// TwinCAT 3 PLC project Plc_Program
// ProgramVersion: 3.1.4026.15
// libraries:
//   CPNTeck - OSCAT BASIC, * (CPNTeck - Automação Industrial)
//   Tc2_MC2, * (Beckhoff Automation GmbH)
//   Tc2_ModbusSrv, * (Beckhoff Automation GmbH)
//   Tc2_Standard, * (Beckhoff Automation GmbH)
//   Tc2_SUPS, * (Beckhoff Automation GmbH)
//   Tc2_System, * (Beckhoff Automation GmbH)
//   Tc2_Utilities, * (Beckhoff Automation GmbH)
// project tree:
//   GVLs/ GVL_Hmi.TcGVL, GVL_Hw.TcGVL, GVL_InterConnection.TcGVL
//   Library/AxisControl/DataTypes/ LAxisCtrl_typeAxisConfig.TcDUT, LAxisCtrl_typeCamIn.TcDUT, LAxisCtrl_typeDiagnostics.TcDUT, LAxisCtrl_typeFastStop.TcDUT, LAxisCtrl_typeGearInAbsolute.TcDUT, LAxisCtrl_typeGearInRelative.TcDUT, LAxisCtrl_typeGeneralSettings.TcDUT, LAxisCtrl_typeHoming.TcDUT, LAxisCtrl_typeJog.TcDUT, LAxisCtrl_typeMoveVelocity.TcDUT, LAxisCtrl_typePhasing.TcDUT, LAxisCtrl_typePosAbsolute.TcDUT, LAxisCtrl_typePosRelative.TcDUT, LAxisCtrl_typePosSuperimposed.TcDUT, LAxisCtrl_typePower.TcDUT, LAxisCtrl_typeStop.TcDUT, LAxisCtrl_typeTorqueLimiting.TcDUT, LRK_typeCamCommand.TcDUT, LRK_typeCamStatus.TcDUT, LRK_typeRotaryKnifeAxisCommand.TcDUT, LRK_typeUsersInterface.TcDUT, MC_SYNCHRONIZEDMOTIONSIMULATION.TcPOU, TO_Cam_Struct_PointData.TcDUT, TO_Cam_Struct_SegmentData.TcDUT
//   Library/AxisControl/ FB_ComplexAxisControl.TcPOU (excluded from build), FB_SimpleAxisControl.TcPOU, MC_TORQUELIMITING.TcPOU
//   Library/Beckhoff/CX9020/ FB_SavePersistentData.TcPOU
//   Library/Beckhoff/EL1008/DataTypes/ EL1008_DEV_CONFIG.TcDUT, EL1008_HWTOPLC_PDOS.TcDUT, EL1008_PDOS.TcDUT
//   Library/Beckhoff/EL1008/ FB_EL1008.TcPOU
//   Library/Beckhoff/EL1809/DataTypes/ EL1809_DEV_CONFIG.TcDUT, EL1809_HWTOPLC_PDOS.TcDUT, EL1809_PDOS.TcDUT
//   Library/Beckhoff/EL1809/ FB_EL1809.TcPOU
//   Library/Beckhoff/EL2809/DataTypes/ EL2809_DEV_CONFIG.TcDUT, EL2809_PDOS.TcDUT, EL2809_PLCTOHW_PDOS.TcDUT
//   Library/Beckhoff/EL2809/ FB_EL2809.TcPOU
//   Library/Beckhoff/EL3002 - Ai 2 x 10V - 12bit/DataTypes/ EL3002_CHANNEL.TcDUT, EL3002_DEV_CONFIG.TcDUT, EL3002_DEV_STATUS.TcDUT, EL3002_HWTOPLC_PDOS.TcDUT, EL3002_PDOS.TcDUT
//   Library/Beckhoff/EL3002 - Ai 2 x 10V - 12bit/ FB_EL3002.TcPOU
//   Library/Beckhoff/EL4004 - AQ 4 x 0-10V/DataTypes/ EL4004_DEV_CONFIG.TcDUT, EL4004_HWTOPLC_PDOS.TcDUT, EL4004_PDOS.TcDUT
//   Library/Beckhoff/EL4004 - AQ 4 x 0-10V/ FB_EL4004.TcPOU
//   Library/Beckhoff/EL5152 -2 x  Encoder Input/DataTypes/ EL5152_CONTROL.TcDUT, EL5152_DEV_CONFIG.TcDUT, EL5152_HWTOPLC.TcDUT, EL5152_HWTOPLC_PDOS.TcDUT, EL5152_PLCTOHW.TcDUT, EL5152_PLCTOHW_PDOS.TcDUT, EL5152_STATUS.TcDUT
//   Library/Beckhoff/EL5152 -2 x  Encoder Input/ FB_EL5152.TcPOU
//   Library/EL6910 - TwinSAFE PLC/ EL6910_ESTOP.TcDUT, EL6910_ESTOP_DIGNOSTICS.TcDUT, EL6910_ESTOP_STATUS.TcDUT, EL6910_HWTOPLC_PDOS.TcDUT, EL6910_PDOS.TcDUT, EL6910_PLCTOHW_PDOS.TcDUT, FB_EL6910.TcPOU
//   Library/FAS/IO-Link/006B51 - IO-Link Master/DataTypes/ _006B51_Channel_State.TcDUT, _006B51_HWTOPLC_PDOS.TcDUT
//   Library/FAS/IO-Link/006B51 - IO-Link Master/ _FB_006B51.TcPOU
//   Library/FAS/IO-Link/00BE31 - IP67 16Di or 16Do/DataTypes/ _00BE31_HWTOPLC_PDOS.TcDUT, _00BE31_PLCTOHW_PDOS.TcDUT
//   Library/FAS/IO-Link/00BE31 - IP67 16Di or 16Do/ _FB_00BE31.TcPOU
//   Library/FAS/IO-Link/00BH11 - 16Di or 16Do/DataTypes/ _00BH11_HWTOPLC_PDOS.TcDUT, _00BH11_PLCTOHW_PDOS.TcDUT
//   Library/FAS/IO-Link/00BH11 - 16Di or 16Do/ _FB_00BH11.TcPOU
//   Library/FAS/IO-Link/00BW12 - 16 Solenoid Island/DataTypes/ _00BW12_PLCTOHW_PDOS.TcDUT
//   Library/FAS/IO-Link/00BW12 - 16 Solenoid Island/ _FB_00BW1.TcPOU
//   Library/FAS/IO-Link/0AC001 - Analog Input/DataTypes/ _0AC001_DEV_CONFIG.TcDUT, _0AC001_HWTOPLC_PDOS.TcDUT
//   Library/FAS/IO-Link/0AC001 - Analog Input/ _FB_0AC001.TcPOU
//   Library/Machine/DryEnd/Alarm Control/ FB_AlarmControl.TcPOU
//   Library/Machine/DryEnd/AutomaticOrderChange/ aocConfig_TypeStruct.TcDUT, aocHmiCommands_TypeStruct.TcDUT, aocHmiStatus_TypeStruct.TcDUT, FB_AutomaticOrderChange.TcPOU, FB_AutomaticOrderChange_V1.TcPOU, FB_AutomaticOrderChange_V1_BAK.TcPOU, lineControlHmiCommands_TypeStruct.TcDUT
//   Library/Machine/DryEnd/Hmi/ hmiAlarms_TypeStruct.TcDUT, hmiCommands_TypeStruct.TcDUT, hmiStatus_TypeStruct.TcDUT, machineConfig_TypeStruct.TcDUT
//   Library/Machine/DryEnd/Order control/DataTypes/ generatedOrderStatusWord_TypeStruct.TcDUT, generatedOrder_TypeStruct.TcDUT, orderConfig_TypeStruct.TcDUT, orderHmiCommands_TypeStruct.TcDUT, orderHmiStatus_TypeStruct.TcDUT, orderVariables_TypeStruct.TcDUT, order_TypeStruct.TcDUT, sheetTypeEnum.TcDUT
//   Library/Machine/DryEnd/Order control/ FB_MetricsAndCalculation.TcPOU
//   Library/Machine/Rotary knife/Config/ rotaryKnifeConfig_TypeStruct.TcDUT, rotaryKnifeHmiStatus_TypeStruct.TcDUT, rotaryKnifeSpeedCurve_TypeConfig.TcDUT, rotaryKnifeStatusWord1_TypeStruct.TcDUT, rotaryKnifeStatusWord2_TypeStruct.TcDUT
//   Library/Machine/Rotary knife/Function Block/ FB_RotaryKnife.TcPOU, FB_RotaryKnife_1.TcPOU, FB_SpeedLimit.TcPOU
//   Library/Machine/Rotary knife/Hmi/ hmiAlarmsRotaryKnife_TypeStruct.TcDUT, rotaryKnifeCommands_TypeStruct.TcDUT, rotaryKnifeStatus_TypeStruct.TcDUT
//   Library/Machine/Slitter/DataTypes/Hmi/ E_LevelSelector.TcDUT, hmiAlarmsSlitter_TypeStruct.TcDUT, hmiCommandsFlaps_TypeStruct.TcDUT, hmiCommandsJog_TypeStruct.TcDUT, hmiCommandsSmallPosCorrection_TypeStruct.TcDUT, hmiSlitterAlarms_TypeStruct.TcDUT, slitterCommands_TypeStruct.TcDUT, slitterConfig_TypeStruct.TcDUT, slitterStatus_TypeStruct.TcDUT
//   Library/Machine/Slitter/FunctionBlocks/ FB_KnifeLubrification.TcPOU, FB_KnifeSharpening.TcPOU, FB_KnifeSharpening_old.TcPOU, FB_PaperDirectionControl.TcPOU, FB_PaperDirectionControl_.TcPOU, FB_PositionsGeneration.TcPOU, FB_ScorerHeight.TcPOU, FB_SlitterControl.TcPOU, FB_SpeedMeter.TcPOU
//   Library/Machine/Stacker/Cpx/ FB_ComplexSheetStackerControl_1.TcPOU, FB_ComplexSheetStackerControl.TcPOU
//   Library/Machine/Stacker/Simple/DataTypes/ hmiAlarmsSimpleStacker_TypeStruct.TcDUT, hmiCommandsSimpleStacker_TypeStruct.TcDUT, hmiStatusSimpleStacker_TypeStruct.TcDUT, SimpleStackerConfig_TypeStruct.TcDUT, SimpleStackerConfig_TypeStruct_1.TcDUT
//   Library/Machine/Stacker/Cpx/DataTypes/ ComplexStackerConfig_TypeStruct.TcDUT, hmiAlarmsComplexStacker_TypeStruct.TcDUT, hmiCommandsComplexStacker_TypeStruct.TcDUT, hmiStatusComplexStacker_TypeStruct.TcDUT
//   Library/Machine/Stacker/Simple/ E_BackstopState.TcDUT, E_ConveyorLevelerState.TcDUT, E_PackageSeparationState.TcDUT, E_SheetStackDischargeState.TcDUT, E_SyncConveyorsState.TcDUT, FB_SimpleSheetStackerControl.TcPOU, FB_SimpleSheetStackerControl_1.TcPOU, FB_SimpleSheetStackerControl_2.TcPOU (not stored), FB_SimpleSheetStackerControl_3.TcPOU
//   Library/Ramp/ FB_Gen_SRamp.TcPOU
//   Library/Sick/DT35-B15251 - Laser Sensor/DataTypes/ _DT35B15251_DEV_CONFIG.TcDUT, _DT35B15251_HWTOPLC_PDOS.TcDUT
//   Library/Sick/DT35-B15251 - Laser Sensor/ _FB_DT35_B15251.TcPOU
//   Library/Inovance/IS620P-CO/DataTypes/ E_IS620P_CO_STATE.TcDUT, IS620P_CO_DEV_CONFIG.TcDUT, IS620P_CO_HWTOPLC_PDOS.TcDUT, IS620P_CO_PLCTOHW_PDOS.TcDUT, IS620P_CO_STATUS.TcDUT
//   Library/Inovance/IS620P-CO/FB/ FB_IS620P_CO.TcPOU
//   / PlcFastTask.TcTTO, PlcTask.TcTTO, RecipeManager.TcRMO (not stored)
//   POUs/ FAST.TcPOU, MAIN.TcPOU
// real-time tasks:
//   TASK PlcTask: cycle T#20ms, priority 20, ADS port 350
//   TASK PlcFastTask: cycle T#5ms, priority 1, ADS port 351
// motion (NC):
//   TASK NC-Task 1 SAF: cycle T#4ms, priority 4, ADS port 501
//   TASK NC-Task 1 SVB: cycle T#10ms, priority 8, ADS port 511
//   AXIS knife1_Axis (id 1)
//     Velo: RefSearch=20, RefSync=2
//     PositionAreaControl: Enable=false
//     OtherSettings: AllowMotionCmdToSlave=true
//     encoder EncType=19
//       EncPara: ScaleFactorNumerator=5.96046448e-07, ModuloFactor=5, Inverse=true, MaxCount=#xffffffff
//         SoftEndMinControl: Enable=true
//         SoftEndMaxControl: Enable=true, Range=950
//         Inc: RefSearchInverse=true, RefSyncInverse=false
//     drive DrvType=16
//       DrvPara: Inverse=true, MaxCount=#xffffffff, DriveControlDWord=#x00020000
//         Analog: TorqueSetpointScale=10, ScaleFactorActTorque=0.1
//         TimeComp: TaskDelayCycles=1
//     controller CtrType=1
//       CtrPara: PriorControlFactor=1
//         PosDiffControl: Enable=false
//         Observer: BandWidth=20
//   AXIS knife2_Axis (id 2)
//     Velo: RefSearch=20, RefSync=2
//     PositionAreaControl: Enable=false
//     OtherSettings: AllowMotionCmdToSlave=true
//     encoder EncType=19
//       EncPara: ScaleFactorNumerator=5.96046448e-07, ModuloFactor=5, Inverse=true, MaxCount=#xffffffff
//         SoftEndMinControl: Enable=true
//         SoftEndMaxControl: Enable=true, Range=1080
//         Inc: RefSearchInverse=true, RefSyncInverse=false
//     drive DrvType=16
//       DrvPara: Inverse=true, MaxCount=#xffffffff, DriveControlDWord=#x00020000
//         Analog: TorqueSetpointScale=10, ScaleFactorActTorque=0.1
//         TimeComp: TaskDelayCycles=1
//     controller CtrType=1
//       CtrPara: PriorControlFactor=1
//         PosDiffControl: Enable=false
//         Observer: BandWidth=20
//   AXIS knife3_Axis (id 3)
//     Velo: RefSearch=20, RefSync=2
//     PositionAreaControl: Enable=false
//     OtherSettings: AllowMotionCmdToSlave=true
//     encoder EncType=19
//       EncPara: ScaleFactorNumerator=5.96046448e-07, ModuloFactor=5, Inverse=true, MaxCount=#xffffffff
//         SoftEndMinControl: Enable=true
//         SoftEndMaxControl: Enable=true, Range=1220
//         Inc: RefSearchInverse=true, RefSyncInverse=false
//     drive DrvType=16
//       DrvPara: Inverse=true, MaxCount=#xffffffff, DriveControlDWord=#x00020000
//         Analog: TorqueSetpointScale=10, ScaleFactorActTorque=0.1
//         TimeComp: TaskDelayCycles=1
//     controller CtrType=1
//       CtrPara: PriorControlFactor=1
//         PosDiffControl: Enable=false
//         Observer: BandWidth=20
//   AXIS knife4_Axis (id 4)
//     Velo: RefSearch=20, RefSync=2
//     PositionAreaControl: Enable=false
//     OtherSettings: AllowMotionCmdToSlave=true
//     encoder EncType=19
//       EncPara: ScaleFactorNumerator=5.96046448e-07, ModuloFactor=5, MaxCount=#xffffffff
//         SoftEndMinControl: Enable=true, Range=1176
//         SoftEndMaxControl: Enable=true, Range=3000
//     drive DrvType=16
//       DrvPara: MaxCount=#xffffffff, DriveControlDWord=#x00020000
//         Analog: TorqueSetpointScale=10, ScaleFactorActTorque=0.1
//         TimeComp: TaskDelayCycles=1
//     controller CtrType=1
//       CtrPara: PriorControlFactor=1
//         PosDiffControl: Enable=false
//         Observer: BandWidth=20
//   AXIS knife5_Axis (id 5)
//     Velo: RefSearch=20, RefSync=2
//     PositionAreaControl: Enable=false
//     OtherSettings: AllowMotionCmdToSlave=true
//     encoder EncType=19
//       EncPara: ScaleFactorNumerator=5.96046448e-07, ModuloFactor=5, MaxCount=#xffffffff
//         SoftEndMinControl: Enable=true, Range=1300
//         SoftEndMaxControl: Enable=true, Range=3000
//     drive DrvType=16
//       DrvPara: MaxCount=#xffffffff, DriveControlDWord=#x00020000
//         Analog: TorqueSetpointScale=10, ScaleFactorActTorque=0.1
//         TimeComp: TaskDelayCycles=1
//     controller CtrType=1
//       CtrPara: PriorControlFactor=1
//         PosDiffControl: Enable=false
//         Observer: BandWidth=20
//   AXIS Scorer1_Axis (id 6)
//     Velo: RefSearch=20, RefSync=2
//     PositionAreaControl: Enable=false
//     OtherSettings: AllowMotionCmdToSlave=true
//     encoder EncType=19
//       EncPara: ScaleFactorNumerator=5.96046448e-07, ModuloFactor=5, Inverse=true, MaxCount=#xffffffff
//         SoftEndMaxControl: Range=968
//         Inc: RefSearchInverse=true, RefSyncInverse=false
//     drive DrvType=16
//       DrvPara: Inverse=true, MaxCount=#xffffffff, DriveControlDWord=#x00020000
//         Analog: TorqueSetpointScale=10, ScaleFactorActTorque=0.1
//         TimeComp: TaskDelayCycles=1
//     controller CtrType=1
//       CtrPara: PriorControlFactor=1
//         PosDiffControl: Enable=false
//         Observer: BandWidth=20
//   AXIS Scorer2_Axis (id 7)
//     Velo: RefSearch=20, RefSync=2
//     PositionAreaControl: Enable=false
//     OtherSettings: AllowMotionCmdToSlave=true
//     encoder EncType=19
//       EncPara: ScaleFactorNumerator=5.96046448e-07, ModuloFactor=5, Inverse=true, MaxCount=#xffffffff
//         SoftEndMaxControl: Range=968
//         Inc: RefSearchInverse=true, RefSyncInverse=false
//     drive DrvType=16
//       DrvPara: Inverse=true, MaxCount=#xffffffff, DriveControlDWord=#x00020000
//         Analog: TorqueSetpointScale=10, ScaleFactorActTorque=0.1
//         TimeComp: TaskDelayCycles=1
//     controller CtrType=1
//       CtrPara: PriorControlFactor=1
//         PosDiffControl: Enable=false
//         Observer: BandWidth=20
//   AXIS Scorer3_Axis (id 8)
//     Velo: RefSearch=20, RefSync=2
//     PositionAreaControl: Enable=false
//     OtherSettings: AllowMotionCmdToSlave=true
//     encoder EncType=19
//       EncPara: ScaleFactorNumerator=5.96046448e-07, ModuloFactor=5, Inverse=true, MaxCount=#xffffffff
//         SoftEndMinControl: Range=364
//         SoftEndMaxControl: Range=1120
//         Inc: RefSearchInverse=true, RefSyncInverse=false
//     drive DrvType=16
//       DrvPara: Inverse=true, MaxCount=#xffffffff, DriveControlDWord=#x00020000
//         Analog: TorqueSetpointScale=10, ScaleFactorActTorque=0.1
//         TimeComp: TaskDelayCycles=1
//     controller CtrType=1
//       CtrPara: PriorControlFactor=1
//         PosDiffControl: Enable=false
//         Observer: BandWidth=20
//   AXIS Scorer4_Axis (id 9)
//     Velo: RefSearch=20, RefSync=2
//     PositionAreaControl: Enable=false
//     OtherSettings: AllowMotionCmdToSlave=true
//     encoder EncType=19
//       EncPara: ScaleFactorNumerator=5.96046448e-07, ModuloFactor=5, Inverse=true, MaxCount=#xffffffff
//         SoftEndMinControl: Range=340
//         SoftEndMaxControl: Range=1120
//         Inc: RefSearchInverse=true, RefSyncInverse=false
//     drive DrvType=16
//       DrvPara: Inverse=true, MaxCount=#xffffffff, DriveControlDWord=#x00020000
//         Analog: TorqueSetpointScale=10, ScaleFactorActTorque=0.1
//         TimeComp: TaskDelayCycles=1
//     controller CtrType=1
//       CtrPara: PriorControlFactor=1
//         PosDiffControl: Enable=false
//         Observer: BandWidth=20
//   AXIS Scorer5_Axis (id 10)
//     Velo: RefSearch=20, RefSync=2
//     PositionAreaControl: Enable=false
//     OtherSettings: AllowMotionCmdToSlave=true
//     encoder EncType=19
//       EncPara: ScaleFactorNumerator=5.96046448e-07, ModuloFactor=5, MaxCount=#xffffffff
//         SoftEndMinControl: Range=1050
//         SoftEndMaxControl: Range=1846
//     drive DrvType=16
//       DrvPara: MaxCount=#xffffffff, DriveControlDWord=#x00020000
//         Analog: TorqueSetpointScale=10, ScaleFactorActTorque=0.1
//         TimeComp: TaskDelayCycles=1
//     controller CtrType=1
//       CtrPara: PriorControlFactor=1
//         PosDiffControl: Enable=false
//         Observer: BandWidth=20
//   AXIS Scorer6_Axis (id 11)
//     Velo: RefSearch=20, RefSync=2
//     PositionAreaControl: Enable=false
//     OtherSettings: AllowMotionCmdToSlave=true
//     encoder EncType=19
//       EncPara: ScaleFactorNumerator=5.96046448e-07, ModuloFactor=5, MaxCount=#xffffffff
//         SoftEndMinControl: Range=1130
//         SoftEndMaxControl: Range=1890
//     drive DrvType=16
//       DrvPara: MaxCount=#xffffffff, DriveControlDWord=#x00020000
//         Analog: TorqueSetpointScale=10, ScaleFactorActTorque=0.1
//         TimeComp: TaskDelayCycles=1
//     controller CtrType=1
//       CtrPara: PriorControlFactor=1
//         PosDiffControl: Enable=false
//         Observer: BandWidth=20
//   AXIS Scorer7_Axis (id 12)
//     Velo: RefSearch=20, RefSync=2
//     PositionAreaControl: Enable=false
//     OtherSettings: AllowMotionCmdToSlave=true
//     encoder EncType=19
//       EncPara: ScaleFactorNumerator=5.96046448e-07, ModuloFactor=5, MaxCount=#xffffffff
//         SoftEndMinControl: Range=1220
//         SoftEndMaxControl: Range=3000
//     drive DrvType=16
//       DrvPara: MaxCount=#xffffffff, DriveControlDWord=#x00020000
//         Analog: TorqueSetpointScale=10, ScaleFactorActTorque=0.1
//         TimeComp: TaskDelayCycles=1
//     controller CtrType=1
//       CtrPara: PriorControlFactor=1
//         PosDiffControl: Enable=false
//         Observer: BandWidth=20
//   AXIS Scorer8_Axis (id 13)
//     Velo: RefSearch=20, RefSync=2
//     PositionAreaControl: Enable=false
//     OtherSettings: AllowMotionCmdToSlave=true
//     encoder EncType=19
//       EncPara: ScaleFactorNumerator=5.96046448e-07, ModuloFactor=5, MaxCount=#xffffffff
//         SoftEndMinControl: Range=1240
//         SoftEndMaxControl: Range=3000
//     drive DrvType=16
//       DrvPara: MaxCount=#xffffffff, DriveControlDWord=#x00020000
//         Analog: TorqueSetpointScale=10, ScaleFactorActTorque=0.1
//         TimeComp: TaskDelayCycles=1
//     controller CtrType=1
//       CtrPara: PriorControlFactor=1
//         PosDiffControl: Enable=false, Range=20
//         Observer: BandWidth=20
// I/O:
//   DEVICE ETC, AmsNetId 192.168.30.79.2.1
//     SLT1+P1=050-BC1 [EK1200-5000 EtherCAT Power supply (2A E-Bus)]
//       SLT1+P1=050-DI1 [EL1809 16Ch. Dig. Input 24V, 3ms]
//       SLT1+P1=050-DI2 [EL1809 16Ch. Dig. Input 24V, 3ms]
//       SLT1+P1=050-DI3 [EL1809 16Ch. Dig. Input 24V, 3ms]
//       SLT1+P1=050-DI4 [EL1809 16Ch. Dig. Input 24V, 3ms]
//       SLT1+P1=050-DI5 [EL1809 16Ch. Dig. Input 24V, 3ms]
//       SLT1+P1=050-DO1 [EL1809 16Ch. Dig. Input 24V, 3ms]
//       SLT1+P1=050-DO2 [EL2809 16Ch. Dig. Output 24V, 0.5A]
//       SLT1+P1=050-DO3 [EL2809 16Ch. Dig. Output 24V, 0.5A]
//       SLT1+P1=050-DO4 [EL2809 16Ch. Dig. Output 24V, 0.5A]
//       SLT1+P1=050-DO5 [EL2809 16Ch. Dig. Output 24V, 0.5A]
//       SLT1+P1=050-DO6 [EL2809 16Ch. Dig. Output 24V, 0.5A]
//       SLT1+P1=050-DO7 [EL2809 16Ch. Dig. Output 24V, 0.5A]
//       SLT1+P1=050-BC2 [EK1110 EtherCAT extension]
//     SLT1+P1=100-UG01 [SD700_ECAT_V1.2_G]
//     SLT1+P1=100-UG02 [SD700_ECAT_V1.2_G]
//     SLT1+P1=100-UG03 [SD700_ECAT_V1.2_G]
//     SLT1+P1=100-UG04 [SD700_ECAT_V1.2_G]
//     SLT1+P1=100-UG05 [SD700_ECAT_V1.2_G]
//     SLT1+P1=100-UG06 [SD700_ECAT_V1.2_G]
//     SLT1+P1=100-UG07 [SD700_ECAT_V1.2_G]
//     SLT1+P1=100-UG08 [SD700_ECAT_V1.2_G]
//     SLT1+P1=100-UG09 [SD700_ECAT_V1.2_G]
//     SLT1+P1=100-UG10 [SD700_ECAT_V1.2_G]
//     SLT1+P1=100-UG11 [SD700_ECAT_V1.2_G]
//     SLT1+P1=100-UG12 [SD700_ECAT_V1.2_G]
//     SLT1+P1=100-UG13 [SD700_ECAT_V1.2_G]
//     RK+P1=050-BC1 [EK1100 EtherCAT Coupler (2A E-Bus)]
//       RK+P1=050-DI1 [EL1809 16Ch. Dig. Input 24V, 3ms]
//       RK+P1=050-DI2 [EL1008 8Ch. Dig. Input 24V, 3ms]
//       RK+P1=050-DO1 [EL2809 16Ch. Dig. Output 24V, 0.5A]
//       RK+P1=050-DO2 [EL2809 16Ch. Dig. Output 24V, 0.5A]
//       RK+P1=050-AI1 [EL3002 2Ch. Ana. Input +/-10V]
//       RK+P1=050-AO1 [EL4004 4Ch. Ana. Output 0-10V, 12bit]
//       RK+P1=050-AO2 [EL4004 4Ch. Ana. Output 0-10V, 12bit] (disabled)
//       RK+P1=050-BE1 [EL9011 End Terminal]
//     STK+P2=050-BC1 [EK1100 EtherCAT Coupler (2A E-Bus)]
//       STK+P2=050-DI1 [EL1809 16Ch. Dig. Input 24V, 3ms]
//       STK+P2=050-DI2 [EL1809 16Ch. Dig. Input 24V, 3ms]
//       STK+P2=050-DO1 [EL2809 16Ch. Dig. Output 24V, 0.5A]
//       STK+P2=050-DO2 [EL2809 16Ch. Dig. Output 24V, 0.5A]
//       STK+P2=050-ENC1 [EL5152 2Ch. Inc. Encoder]
//       STK+P2=050-AO1 [EL4004 4Ch. Ana. Output 0-10V, 12bit]
//       STK+P2=050-AO2 [EL4004 4Ch. Ana. Output 0-10V, 12bit]
//       STK+P2=050-AO3 [EL4004 4Ch. Ana. Output 0-10V, 12bit]
//       STK+P2=050-AO4 [EL4004 4Ch. Ana. Output 0-10V, 12bit]
//       STK+P2=050-SP1 [EL6910, TwinSAFE PLC]
//       STK+P2=050-SI1 [EL1904, 4 Ch. Safety Input 24V, TwinSAFE]
//         modules: Module 1 (FSOES)
//       STK+P2=050-SI2 [EL1904, 4 Ch. Safety Input 24V, TwinSAFE]
//         modules: Module 1 (FSOES)
//       STK+P2=050-SO1 [EL2904, 4 Ch. Safety Output 24V, 0.5A, TwinSAFE]
//         modules: Module 1 (FSOES), Module 2 (DO)
//       STK+P2=050-BC2 [EL6751 CANopen Master]
//       STK+P2=050-BC3 [EK1110 EtherCAT extension]
//     STK+M=050-BC1 [FNI ECT-504-105-M]
//       modules: STKL+M=050-DIO1 - IO-Link slave IP67 [Machine drive side], STKL+M=050-DIO2  - IO-Link slave IP24 [Lower command box], STKL+M=050-BE1  - IO-Link Sick distance sensor [Backstop], STKU+M=050-DIO1  - IO-Link slave IP24 [Lower command box], STKU+M=050-DIO2  - IO-Link slave IP24 [Uppercommand box], STKU+M=050-DIO3  - IO-Link slave IP24 [Elevator drive side], Module 7 (Digital_IN), Module 8 (Digital_IN)
//   DEVICE Device 3 (NOV-DP-RAM)
//   DEVICE CANopen, AmsNetId 192.168.30.79.3.1
//     STK+P2=100-UG8 - Backstop Servo Drive
//     STK+P2=100-UG8 - Elevator Servo Drive
// variable links:
//   ETC <-> ETC/STK+P2=050-BC1/STK+P2=050-SI2
//     STK+P2=050-BC1/STK+P2=050-SP1/ConnectionOutputs/Message_4 RxPDO <-> Module 1 (FSOES)/TxPDO/FSOE
//   ETC <-> ETC/STK+P2=050-BC1/STK+P2=050-SO1
//     STK+P2=050-BC1/STK+P2=050-SP1/ConnectionOutputs/Message_5 RxPDO <-> Module 1 (FSOES)/TxPDO/FSOE
//   ETC <-> ETC/STK+P2=050-BC1/STK+P2=050-SP1
//     STK+P2=050-BC1/STK+P2=050-SI1/Module 1 (FSOES)/RxPDO/FSOE <-> ConnectionInputs/Message_3 TxPDO
//     STK+P2=050-BC1/STK+P2=050-SI2/Module 1 (FSOES)/RxPDO/FSOE <-> ConnectionInputs/Message_4 TxPDO
//     STK+P2=050-BC1/STK+P2=050-SI1/Module 1 (FSOES)/TxPDO/FSOE <-> ConnectionOutputs/Message_3 RxPDO
//     STK+P2=050-BC1/STK+P2=050-SO1/Module 1 (FSOES)/RxPDO/FSOE <-> ConnectionInputs/Message_5 TxPDO
//   NC-Task 1 SAF/Axes/Scorer1_Axis <-> ETC/SLT1+P1=100-UG06
//     Drive/Inputs/In/nDcOutputTime <-> InfoData/DcOutputShift
//     Drive/Inputs/In/nState1 <-> 2nd TxPDO Mapping/Status Word
//     Drive/Inputs/In/nState2 <-> 2nd TxPDO Mapping/Status Word @bit 8
//     Drive/Inputs/In/nState4 @bit 1 <-> WcState/InputToggle
//     Drive/Inputs/In/nState4 <-> WcState/WcState
//     Drive/Outputs/Out/nCtrl1 <-> 2nd RxPDO Mapping/Control Word
//     Drive/Outputs/Out/nCtrl2 <-> 2nd RxPDO Mapping/Control Word @bit 8
//     Drive/Outputs/Out/nDataOut1 <-> 2nd RxPDO Mapping/TargetPosition
//     Drive/Outputs/Out/nDataOut2 <-> 2nd RxPDO Mapping/TargetVelocity
//     Enc/Inputs/In/nDataIn1 <-> 2nd TxPDO Mapping/ActualPosition
//     Enc/Inputs/In/nDataIn7 <-> 2nd TxPDO Mapping/Velocity actual value
//     Enc/Inputs/In/nDcInputTime <-> InfoData/DcInputShift
//     Enc/Inputs/In/nState4 @bit 1 <-> WcState/InputToggle
//     Enc/Inputs/In/nState4 <-> WcState/WcState
//   NC-Task 1 SAF/Axes/Scorer2_Axis <-> ETC/SLT1+P1=100-UG07
//     Drive/Inputs/In/nDcOutputTime <-> InfoData/DcOutputShift
//     Drive/Inputs/In/nState1 <-> 2nd TxPDO Mapping/Status Word
//     Drive/Inputs/In/nState2 <-> 2nd TxPDO Mapping/Status Word @bit 8
//     Drive/Inputs/In/nState4 @bit 1 <-> WcState/InputToggle
//     Drive/Inputs/In/nState4 <-> WcState/WcState
//     Drive/Outputs/Out/nCtrl1 <-> 2nd RxPDO Mapping/Control Word
//     Drive/Outputs/Out/nCtrl2 <-> 2nd RxPDO Mapping/Control Word @bit 8
//     Drive/Outputs/Out/nDataOut1 <-> 2nd RxPDO Mapping/TargetPosition
//     Drive/Outputs/Out/nDataOut2 <-> 2nd RxPDO Mapping/TargetVelocity
//     Enc/Inputs/In/nDataIn1 <-> 2nd TxPDO Mapping/ActualPosition
//     Enc/Inputs/In/nDataIn7 <-> 2nd TxPDO Mapping/Velocity actual value
//     Enc/Inputs/In/nDcInputTime <-> InfoData/DcInputShift
//     Enc/Inputs/In/nState4 @bit 1 <-> WcState/InputToggle
//     Enc/Inputs/In/nState4 <-> WcState/WcState
//   NC-Task 1 SAF/Axes/Scorer3_Axis <-> ETC/SLT1+P1=100-UG08
//     Drive/Inputs/In/nDcOutputTime <-> InfoData/DcOutputShift
//     Drive/Inputs/In/nState1 <-> 2nd TxPDO Mapping/Status Word
//     Drive/Inputs/In/nState2 <-> 2nd TxPDO Mapping/Status Word @bit 8
//     Drive/Inputs/In/nState4 @bit 1 <-> WcState/InputToggle
//     Drive/Inputs/In/nState4 <-> WcState/WcState
//     Drive/Outputs/Out/nCtrl1 <-> 2nd RxPDO Mapping/Control Word
//     Drive/Outputs/Out/nCtrl2 <-> 2nd RxPDO Mapping/Control Word @bit 8
//     Drive/Outputs/Out/nDataOut1 <-> 2nd RxPDO Mapping/TargetPosition
//     Drive/Outputs/Out/nDataOut2 <-> 2nd RxPDO Mapping/TargetVelocity
//     Enc/Inputs/In/nDataIn1 <-> 2nd TxPDO Mapping/ActualPosition
//     Enc/Inputs/In/nDataIn7 <-> 2nd TxPDO Mapping/Velocity actual value
//     Enc/Inputs/In/nDcInputTime <-> InfoData/DcInputShift
//     Enc/Inputs/In/nState4 @bit 1 <-> WcState/InputToggle
//     Enc/Inputs/In/nState4 <-> WcState/WcState
//   NC-Task 1 SAF/Axes/Scorer4_Axis <-> ETC/SLT1+P1=100-UG09
//     Drive/Inputs/In/nDcOutputTime <-> InfoData/DcOutputShift
//     Drive/Inputs/In/nState1 <-> 2nd TxPDO Mapping/Status Word
//     Drive/Inputs/In/nState2 <-> 2nd TxPDO Mapping/Status Word @bit 8
//     Drive/Inputs/In/nState4 @bit 1 <-> WcState/InputToggle
//     Drive/Inputs/In/nState4 <-> WcState/WcState
//     Drive/Outputs/Out/nCtrl1 <-> 2nd RxPDO Mapping/Control Word
//     Drive/Outputs/Out/nCtrl2 <-> 2nd RxPDO Mapping/Control Word @bit 8
//     Drive/Outputs/Out/nDataOut1 <-> 2nd RxPDO Mapping/TargetPosition
//     Drive/Outputs/Out/nDataOut2 <-> 2nd RxPDO Mapping/TargetVelocity
//     Enc/Inputs/In/nDataIn1 <-> 2nd TxPDO Mapping/ActualPosition
//     Enc/Inputs/In/nDataIn7 <-> 2nd TxPDO Mapping/Velocity actual value
//     Enc/Inputs/In/nDcInputTime <-> InfoData/DcInputShift
//     Enc/Inputs/In/nState4 @bit 1 <-> WcState/InputToggle
//     Enc/Inputs/In/nState4 <-> WcState/WcState
//   NC-Task 1 SAF/Axes/Scorer5_Axis <-> ETC/SLT1+P1=100-UG10
//     Drive/Inputs/In/nDcOutputTime <-> InfoData/DcOutputShift
//     Drive/Inputs/In/nState1 <-> 2nd TxPDO Mapping/Status Word
//     Drive/Inputs/In/nState2 <-> 2nd TxPDO Mapping/Status Word @bit 8
//     Drive/Inputs/In/nState4 @bit 1 <-> WcState/InputToggle
//     Drive/Inputs/In/nState4 <-> WcState/WcState
//     Drive/Outputs/Out/nCtrl1 <-> 2nd RxPDO Mapping/Control Word
//     Drive/Outputs/Out/nCtrl2 <-> 2nd RxPDO Mapping/Control Word @bit 8
//     Drive/Outputs/Out/nDataOut1 <-> 2nd RxPDO Mapping/TargetPosition
//     Drive/Outputs/Out/nDataOut2 <-> 2nd RxPDO Mapping/TargetVelocity
//     Enc/Inputs/In/nDataIn1 <-> 2nd TxPDO Mapping/ActualPosition
//     Enc/Inputs/In/nDataIn7 <-> 2nd TxPDO Mapping/Velocity actual value
//     Enc/Inputs/In/nDcInputTime <-> InfoData/DcInputShift
//     Enc/Inputs/In/nState4 @bit 1 <-> WcState/InputToggle
//     Enc/Inputs/In/nState4 <-> WcState/WcState
//   NC-Task 1 SAF/Axes/Scorer6_Axis <-> ETC/SLT1+P1=100-UG11
//     Drive/Inputs/In/nDcOutputTime <-> InfoData/DcOutputShift
//     Drive/Inputs/In/nState1 <-> 2nd TxPDO Mapping/Status Word
//     Drive/Inputs/In/nState2 <-> 2nd TxPDO Mapping/Status Word @bit 8
//     Drive/Inputs/In/nState4 @bit 1 <-> WcState/InputToggle
//     Drive/Inputs/In/nState4 <-> WcState/WcState
//     Drive/Outputs/Out/nCtrl1 <-> 2nd RxPDO Mapping/Control Word
//     Drive/Outputs/Out/nCtrl2 <-> 2nd RxPDO Mapping/Control Word @bit 8
//     Drive/Outputs/Out/nDataOut1 <-> 2nd RxPDO Mapping/TargetPosition
//     Drive/Outputs/Out/nDataOut2 <-> 2nd RxPDO Mapping/TargetVelocity
//     Enc/Inputs/In/nDataIn1 <-> 2nd TxPDO Mapping/ActualPosition
//     Enc/Inputs/In/nDataIn7 <-> 2nd TxPDO Mapping/Velocity actual value
//     Enc/Inputs/In/nDcInputTime <-> InfoData/DcInputShift
//     Enc/Inputs/In/nState4 @bit 1 <-> WcState/InputToggle
//     Enc/Inputs/In/nState4 <-> WcState/WcState
//   NC-Task 1 SAF/Axes/Scorer7_Axis <-> ETC/SLT1+P1=100-UG12
//     Drive/Inputs/In/nDcOutputTime <-> InfoData/DcOutputShift
//     Drive/Inputs/In/nState1 <-> 2nd TxPDO Mapping/Status Word
//     Drive/Inputs/In/nState2 <-> 2nd TxPDO Mapping/Status Word @bit 8
//     Drive/Inputs/In/nState4 @bit 1 <-> WcState/InputToggle
//     Drive/Inputs/In/nState4 <-> WcState/WcState
//     Drive/Outputs/Out/nCtrl1 <-> 2nd RxPDO Mapping/Control Word
//     Drive/Outputs/Out/nCtrl2 <-> 2nd RxPDO Mapping/Control Word @bit 8
//     Drive/Outputs/Out/nDataOut1 <-> 2nd RxPDO Mapping/TargetPosition
//     Drive/Outputs/Out/nDataOut2 <-> 2nd RxPDO Mapping/TargetVelocity
//     Enc/Inputs/In/nDataIn1 <-> 2nd TxPDO Mapping/ActualPosition
//     Enc/Inputs/In/nDataIn7 <-> 2nd TxPDO Mapping/Velocity actual value
//     Enc/Inputs/In/nDcInputTime <-> InfoData/DcInputShift
//     Enc/Inputs/In/nState4 @bit 1 <-> WcState/InputToggle
//     Enc/Inputs/In/nState4 <-> WcState/WcState
//   NC-Task 1 SAF/Axes/Scorer8_Axis <-> ETC/SLT1+P1=100-UG13
//     Drive/Inputs/In/nDcOutputTime <-> InfoData/DcOutputShift
//     Drive/Inputs/In/nState1 <-> 2nd TxPDO Mapping/Status Word
//     Drive/Inputs/In/nState2 <-> 2nd TxPDO Mapping/Status Word @bit 8
//     Drive/Inputs/In/nState4 @bit 1 <-> WcState/InputToggle
//     Drive/Inputs/In/nState4 <-> WcState/WcState
//     Drive/Outputs/Out/nCtrl1 <-> 2nd RxPDO Mapping/Control Word
//     Drive/Outputs/Out/nCtrl2 <-> 2nd RxPDO Mapping/Control Word @bit 8
//     Drive/Outputs/Out/nDataOut1 <-> 2nd RxPDO Mapping/TargetPosition
//     Drive/Outputs/Out/nDataOut2 <-> 2nd RxPDO Mapping/TargetVelocity
//     Enc/Inputs/In/nDataIn1 <-> 2nd TxPDO Mapping/ActualPosition
//     Enc/Inputs/In/nDataIn7 <-> 2nd TxPDO Mapping/Velocity actual value
//     Enc/Inputs/In/nDcInputTime <-> InfoData/DcInputShift
//     Enc/Inputs/In/nState4 @bit 1 <-> WcState/InputToggle
//     Enc/Inputs/In/nState4 <-> WcState/WcState
//   NC-Task 1 SAF/Axes/knife1_Axis <-> ETC/SLT1+P1=100-UG01
//     Drive/Inputs/In/nDcOutputTime <-> InfoData/DcOutputShift
//     Drive/Inputs/In/nState1 <-> 2nd TxPDO Mapping/Status Word
//     Drive/Inputs/In/nState2 <-> 2nd TxPDO Mapping/Status Word @bit 8
//     Drive/Inputs/In/nState4 @bit 1 <-> WcState/InputToggle
//     Drive/Inputs/In/nState4 <-> WcState/WcState
//     Drive/Outputs/Out/nCtrl1 <-> 2nd RxPDO Mapping/Control Word
//     Drive/Outputs/Out/nCtrl2 <-> 2nd RxPDO Mapping/Control Word @bit 8
//     Drive/Outputs/Out/nDataOut1 <-> 2nd RxPDO Mapping/TargetPosition
//     Drive/Outputs/Out/nDataOut2 <-> 2nd RxPDO Mapping/TargetVelocity
//     Enc/Inputs/In/nDataIn1 <-> 2nd TxPDO Mapping/ActualPosition
//     Enc/Inputs/In/nDataIn7 <-> 2nd TxPDO Mapping/Velocity actual value
//     Enc/Inputs/In/nDcInputTime <-> InfoData/DcInputShift
//     Enc/Inputs/In/nState4 @bit 1 <-> WcState/InputToggle
//     Enc/Inputs/In/nState4 <-> WcState/WcState
//   NC-Task 1 SAF/Axes/knife2_Axis <-> ETC/SLT1+P1=100-UG02
//     Drive/Inputs/In/nDcOutputTime <-> InfoData/DcOutputShift
//     Drive/Inputs/In/nState1 <-> 2nd TxPDO Mapping/Status Word
//     Drive/Inputs/In/nState2 <-> 2nd TxPDO Mapping/Status Word @bit 8
//     Drive/Inputs/In/nState4 @bit 1 <-> WcState/InputToggle
//     Drive/Inputs/In/nState4 <-> WcState/WcState
//     Drive/Outputs/Out/nCtrl1 <-> 2nd RxPDO Mapping/Control Word
//     Drive/Outputs/Out/nCtrl2 <-> 2nd RxPDO Mapping/Control Word @bit 8
//     Drive/Outputs/Out/nDataOut1 <-> 2nd RxPDO Mapping/TargetPosition
//     Drive/Outputs/Out/nDataOut2 <-> 2nd RxPDO Mapping/TargetVelocity
//     Enc/Inputs/In/nDataIn1 <-> 2nd TxPDO Mapping/ActualPosition
//     Enc/Inputs/In/nDataIn7 <-> 2nd TxPDO Mapping/Velocity actual value
//     Enc/Inputs/In/nDcInputTime <-> InfoData/DcInputShift
//     Enc/Inputs/In/nState4 @bit 1 <-> WcState/InputToggle
//     Enc/Inputs/In/nState4 <-> WcState/WcState
//   NC-Task 1 SAF/Axes/knife3_Axis <-> ETC/SLT1+P1=100-UG03
//     Drive/Inputs/In/nDcOutputTime <-> InfoData/DcOutputShift
//     Drive/Inputs/In/nState1 <-> 2nd TxPDO Mapping/Status Word
//     Drive/Inputs/In/nState2 <-> 2nd TxPDO Mapping/Status Word @bit 8
//     Drive/Inputs/In/nState4 @bit 1 <-> WcState/InputToggle
//     Drive/Inputs/In/nState4 <-> WcState/WcState
//     Drive/Outputs/Out/nCtrl1 <-> 2nd RxPDO Mapping/Control Word
//     Drive/Outputs/Out/nCtrl2 <-> 2nd RxPDO Mapping/Control Word @bit 8
//     Drive/Outputs/Out/nDataOut1 <-> 2nd RxPDO Mapping/TargetPosition
//     Drive/Outputs/Out/nDataOut2 <-> 2nd RxPDO Mapping/TargetVelocity
//     Enc/Inputs/In/nDataIn1 <-> 2nd TxPDO Mapping/ActualPosition
//     Enc/Inputs/In/nDataIn7 <-> 2nd TxPDO Mapping/Velocity actual value
//     Enc/Inputs/In/nDcInputTime <-> InfoData/DcInputShift
//     Enc/Inputs/In/nState4 @bit 1 <-> WcState/InputToggle
//     Enc/Inputs/In/nState4 <-> WcState/WcState
//   NC-Task 1 SAF/Axes/knife4_Axis <-> ETC/SLT1+P1=100-UG04
//     Drive/Inputs/In/nDcOutputTime <-> InfoData/DcOutputShift
//     Drive/Inputs/In/nState1 <-> 2nd TxPDO Mapping/Status Word
//     Drive/Inputs/In/nState2 <-> 2nd TxPDO Mapping/Status Word @bit 8
//     Drive/Inputs/In/nState4 @bit 1 <-> WcState/InputToggle
//     Drive/Inputs/In/nState4 <-> WcState/WcState
//     Drive/Outputs/Out/nCtrl1 <-> 2nd RxPDO Mapping/Control Word
//     Drive/Outputs/Out/nCtrl2 <-> 2nd RxPDO Mapping/Control Word @bit 8
//     Drive/Outputs/Out/nDataOut1 <-> 2nd RxPDO Mapping/TargetPosition
//     Drive/Outputs/Out/nDataOut2 <-> 2nd RxPDO Mapping/TargetVelocity
//     Enc/Inputs/In/nDataIn1 <-> 2nd TxPDO Mapping/ActualPosition
//     Enc/Inputs/In/nDataIn7 <-> 2nd TxPDO Mapping/Velocity actual value
//     Enc/Inputs/In/nDcInputTime <-> InfoData/DcInputShift
//     Enc/Inputs/In/nState4 @bit 1 <-> WcState/InputToggle
//     Enc/Inputs/In/nState4 <-> WcState/WcState
//   NC-Task 1 SAF/Axes/knife5_Axis <-> ETC/SLT1+P1=100-UG05
//     Drive/Inputs/In/nDcOutputTime <-> InfoData/DcOutputShift
//     Drive/Inputs/In/nState1 <-> 2nd TxPDO Mapping/Status Word
//     Drive/Inputs/In/nState2 <-> 2nd TxPDO Mapping/Status Word @bit 8
//     Drive/Inputs/In/nState4 @bit 1 <-> WcState/InputToggle
//     Drive/Inputs/In/nState4 <-> WcState/WcState
//     Drive/Outputs/Out/nCtrl1 <-> 2nd RxPDO Mapping/Control Word
//     Drive/Outputs/Out/nCtrl2 <-> 2nd RxPDO Mapping/Control Word @bit 8
//     Drive/Outputs/Out/nDataOut1 <-> 2nd RxPDO Mapping/TargetPosition
//     Drive/Outputs/Out/nDataOut2 <-> 2nd RxPDO Mapping/TargetVelocity
//     Enc/Inputs/In/nDataIn1 <-> 2nd TxPDO Mapping/ActualPosition
//     Enc/Inputs/In/nDataIn7 <-> 2nd TxPDO Mapping/Velocity actual value
//     Enc/Inputs/In/nDcInputTime <-> InfoData/DcInputShift
//     Enc/Inputs/In/nState4 @bit 1 <-> WcState/InputToggle
//     Enc/Inputs/In/nState4 <-> WcState/WcState
//   Plc_Program/Plc_Program Instance <-> CANopen/STK+P2=100-UG8 - Backstop Servo Drive
//     PlcTask Inputs/.STKU_P2_100_UG8.HwToPlc/actualPosition <-> TxPDO 2 - Feedback/Inputs/ActualPosition_6064
//     PlcTask Inputs/.STKU_P2_100_UG8.HwToPlc/actualVelocity <-> TxPDO 2 - Feedback/Inputs/ActualVelocity_606C
//     PlcTask Inputs/.STKU_P2_100_UG8.HwToPlc/diagFlag <-> Inputs/DiagFlag
//     PlcTask Inputs/.STKU_P2_100_UG8.HwToPlc/modeDisplay <-> TxPDO 1 - Status/Inputs/ModeDisplay_6061
//     PlcTask Inputs/.STKU_P2_100_UG8.HwToPlc/nodeState <-> Inputs/NodeState
//     PlcTask Inputs/.STKU_P2_100_UG8.HwToPlc/statusWord <-> TxPDO 1 - Status/Inputs/StatusWord_6041
//     PlcTask Outputs/.STKU_P2_100_UG8.PlcToHw/controlWord <-> RxPDO 1 - Control/Outputs/ControlWord_6040
//     PlcTask Outputs/.STKU_P2_100_UG8.PlcToHw/modeCommand <-> RxPDO 1 - Control/Outputs/ModeCommand_6060
//     PlcTask Outputs/.STKU_P2_100_UG8.PlcToHw/profileAcceleration <-> RxPDO 3 - Acceleration and deceleration/Outputs/ProfileAcceleration_6083
//     PlcTask Outputs/.STKU_P2_100_UG8.PlcToHw/profileDeceleration <-> RxPDO 3 - Acceleration and deceleration/Outputs/ProfileDeceleration_6084
//     PlcTask Outputs/.STKU_P2_100_UG8.PlcToHw/profileVelocity <-> RxPDO 2 - Position profile/Outputs/ProfileVelocity_6081
//     PlcTask Outputs/.STKU_P2_100_UG8.PlcToHw/targetPosition <-> RxPDO 2 - Position profile/Outputs/TargetPosition_607A
//     PlcTask Outputs/.STKU_P2_100_UG8.PlcToHw/targetVelocity <-> RxPDO 4 - Velocity reference/Outputs/TargetVelocity_60FF
//   Plc_Program/Plc_Program Instance <-> CANopen/STK+P2=100-UG8 - Elevator Servo Drive
//     PlcTask Inputs/.STKU_P2_100_UG9.HwToPlc/actualPosition <-> TxPDO 2 - Feedback/Inputs/ActualPosition_6064
//     PlcTask Inputs/.STKU_P2_100_UG9.HwToPlc/actualVelocity <-> TxPDO 2 - Feedback/Inputs/ActualVelocity_606C
//     PlcTask Inputs/.STKU_P2_100_UG9.HwToPlc/diagFlag <-> Inputs/DiagFlag
//     PlcTask Inputs/.STKU_P2_100_UG9.HwToPlc/modeDisplay <-> TxPDO 1 - Status/Inputs/ModeDisplay_6061
//     PlcTask Inputs/.STKU_P2_100_UG9.HwToPlc/nodeState <-> Inputs/NodeState
//     PlcTask Inputs/.STKU_P2_100_UG9.HwToPlc/statusWord <-> TxPDO 1 - Status/Inputs/StatusWord_6041
//     PlcTask Outputs/.STKU_P2_100_UG9.PlcToHw/controlWord <-> RxPDO 1 - Control/Outputs/ControlWord_6040
//     PlcTask Outputs/.STKU_P2_100_UG9.PlcToHw/modeCommand <-> RxPDO 1 - Control/Outputs/ModeCommand_6060
//     PlcTask Outputs/.STKU_P2_100_UG9.PlcToHw/profileAcceleration <-> RxPDO 3 - Acceleration and deceleration/Outputs/ProfileAcceleration_6083
//     PlcTask Outputs/.STKU_P2_100_UG9.PlcToHw/profileDeceleration <-> RxPDO 3 - Acceleration and deceleration/Outputs/ProfileDeceleration_6084
//     PlcTask Outputs/.STKU_P2_100_UG9.PlcToHw/profileVelocity <-> RxPDO 2 - Position profile/Outputs/ProfileVelocity_6081
//     PlcTask Outputs/.STKU_P2_100_UG9.PlcToHw/targetPosition <-> RxPDO 2 - Position profile/Outputs/TargetPosition_607A
//     PlcTask Outputs/.STKU_P2_100_UG9.PlcToHw/targetVelocity <-> RxPDO 4 - Velocity reference/Outputs/TargetVelocity_60FF
//   Plc_Program/Plc_Program Instance <-> ETC/RK+P1=050-BC1/RK+P1=050-AI1
//     PlcFastTask Inputs/.ARK_P1_050_AI01.PDOS.HwToPLC.Channel1/Status/Error <-> AI Standard Channel 1/Status/Error
//     PlcFastTask Inputs/.ARK_P1_050_AI01.PDOS.HwToPLC.Channel2/Status/Error <-> AI Standard Channel 2/Status/Error
//     PlcFastTask Inputs/.ARK_P1_050_AI01.PDOS.HwToPLC.Channel1/Status/Overrange <-> AI Standard Channel 1/Status/Overrange
//     PlcFastTask Inputs/.ARK_P1_050_AI01.PDOS.HwToPLC.Channel2/Status/Overrange <-> AI Standard Channel 2/Status/Overrange
//     PlcFastTask Inputs/.ARK_P1_050_AI01.PDOS.HwToPLC.Channel1/Status/Underrange <-> AI Standard Channel 1/Status/Underrange
//     PlcFastTask Inputs/.ARK_P1_050_AI01.PDOS.HwToPLC.Channel2/Status/Underrange <-> AI Standard Channel 2/Status/Underrange
//     PlcFastTask Inputs/.ARK_P1_050_AI01.PDOS.HwToPLC.Channel1/Value <-> AI Standard Channel 1/Value
//     PlcFastTask Inputs/.ARK_P1_050_AI01.PDOS.HwToPLC.Channel2/Value <-> AI Standard Channel 2/Value
//   Plc_Program/Plc_Program Instance <-> ETC/RK+P1=050-BC1/RK+P1=050-AO1
//     PlcFastTask Outputs/.ARK_P1_050_AO01.PDOS.HwToPLC.Channel1 <-> AO Outputs Channel 1/Analog output
//     PlcFastTask Outputs/.ARK_P1_050_AO01.PDOS.HwToPLC.Channel2 <-> AO Outputs Channel 2/Analog output
//     PlcFastTask Outputs/.ARK_P1_050_AO01.PDOS.HwToPLC.Channel3 <-> AO Outputs Channel 3/Analog output
//     PlcFastTask Outputs/.ARK_P1_050_AO01.PDOS.HwToPLC.Channel4 <-> AO Outputs Channel 4/Analog output
//   Plc_Program/Plc_Program Instance <-> ETC/RK+P1=050-BC1/RK+P1=050-AO2
//     PlcFastTask Outputs/.ARK_P1_050_AO02.PDOS.HwToPLC.Channel1 <-> AO Outputs Channel 1/Analog output
//     PlcFastTask Outputs/.ARK_P1_050_AO02.PDOS.HwToPLC.Channel2 <-> AO Outputs Channel 2/Analog output
//     PlcFastTask Outputs/.ARK_P1_050_AO02.PDOS.HwToPLC.Channel3 <-> AO Outputs Channel 3/Analog output
//     PlcFastTask Outputs/.ARK_P1_050_AO02.PDOS.HwToPLC.Channel4 <-> AO Outputs Channel 4/Analog output
//   Plc_Program/Plc_Program Instance <-> ETC/RK+P1=050-BC1/RK+P1=050-DI1
//     PlcFastTask Inputs/.ARK_P1_050_DI01.PDOS.digitalInput_00 <-> Channel 1/Input
//     PlcFastTask Inputs/.ARK_P1_050_DI01.PDOS.digitalInput_01 <-> Channel 2/Input
//     PlcFastTask Inputs/.ARK_P1_050_DI01.PDOS.digitalInput_02 <-> Channel 3/Input
//     PlcFastTask Inputs/.ARK_P1_050_DI01.PDOS.digitalInput_03 <-> Channel 4/Input
//     PlcFastTask Inputs/.ARK_P1_050_DI01.PDOS.digitalInput_04 <-> Channel 5/Input
//     PlcFastTask Inputs/.ARK_P1_050_DI01.PDOS.digitalInput_05 <-> Channel 6/Input
//     PlcFastTask Inputs/.ARK_P1_050_DI01.PDOS.digitalInput_06 <-> Channel 7/Input
//     PlcFastTask Inputs/.ARK_P1_050_DI01.PDOS.digitalInput_07 <-> Channel 8/Input
//     PlcFastTask Inputs/.ARK_P1_050_DI01.PDOS.digitalInput_08 <-> Channel 9/Input
//     PlcFastTask Inputs/.ARK_P1_050_DI01.PDOS.digitalInput_09 <-> Channel 10/Input
//     PlcFastTask Inputs/.ARK_P1_050_DI01.PDOS.digitalInput_10 <-> Channel 11/Input
//     PlcFastTask Inputs/.ARK_P1_050_DI01.PDOS.digitalInput_11 <-> Channel 12/Input
//     PlcFastTask Inputs/.ARK_P1_050_DI01.PDOS.digitalInput_12 <-> Channel 13/Input
//     PlcFastTask Inputs/.ARK_P1_050_DI01.PDOS.digitalInput_13 <-> Channel 14/Input
//     PlcFastTask Inputs/.ARK_P1_050_DI01.PDOS.digitalInput_14 <-> Channel 15/Input
//     PlcFastTask Inputs/.ARK_P1_050_DI01.PDOS.digitalInput_15 <-> Channel 16/Input
//   Plc_Program/Plc_Program Instance <-> ETC/RK+P1=050-BC1/RK+P1=050-DO1
//     PlcFastTask Outputs/.ARK_P1_050_DO01.PDOS.PlcToHw.digitalOutput_00 <-> Channel 1/Output
//     PlcFastTask Outputs/.ARK_P1_050_DO01.PDOS.PlcToHw.digitalOutput_01 <-> Channel 2/Output
//     PlcFastTask Outputs/.ARK_P1_050_DO01.PDOS.PlcToHw.digitalOutput_02 <-> Channel 3/Output
//     PlcFastTask Outputs/.ARK_P1_050_DO01.PDOS.PlcToHw.digitalOutput_03 <-> Channel 4/Output
//     PlcFastTask Outputs/.ARK_P1_050_DO01.PDOS.PlcToHw.digitalOutput_04 <-> Channel 5/Output
//     PlcFastTask Outputs/.ARK_P1_050_DO01.PDOS.PlcToHw.digitalOutput_05 <-> Channel 6/Output
//     PlcFastTask Outputs/.ARK_P1_050_DO01.PDOS.PlcToHw.digitalOutput_06 <-> Channel 7/Output
//     PlcFastTask Outputs/.ARK_P1_050_DO01.PDOS.PlcToHw.digitalOutput_07 <-> Channel 8/Output
//     PlcFastTask Outputs/.ARK_P1_050_DO01.PDOS.PlcToHw.digitalOutput_08 <-> Channel 9/Output
//     PlcFastTask Outputs/.ARK_P1_050_DO01.PDOS.PlcToHw.digitalOutput_09 <-> Channel 10/Output
//     PlcFastTask Outputs/.ARK_P1_050_DO01.PDOS.PlcToHw.digitalOutput_10 <-> Channel 11/Output
//     PlcFastTask Outputs/.ARK_P1_050_DO01.PDOS.PlcToHw.digitalOutput_11 <-> Channel 12/Output
//     PlcFastTask Outputs/.ARK_P1_050_DO01.PDOS.PlcToHw.digitalOutput_12 <-> Channel 13/Output
//     PlcFastTask Outputs/.ARK_P1_050_DO01.PDOS.PlcToHw.digitalOutput_13 <-> Channel 14/Output
//     PlcFastTask Outputs/.ARK_P1_050_DO01.PDOS.PlcToHw.digitalOutput_14 <-> Channel 15/Output
//     PlcFastTask Outputs/.ARK_P1_050_DO01.PDOS.PlcToHw.digitalOutput_15 <-> Channel 16/Output
//   Plc_Program/Plc_Program Instance <-> ETC/RK+P1=050-BC1/RK+P1=050-DO2
//     PlcFastTask Outputs/.ARK_P1_050_DO02.PDOS.PlcToHw.digitalOutput_00 <-> Channel 1/Output
//     PlcFastTask Outputs/.ARK_P1_050_DO02.PDOS.PlcToHw.digitalOutput_01 <-> Channel 2/Output
//     PlcFastTask Outputs/.ARK_P1_050_DO02.PDOS.PlcToHw.digitalOutput_02 <-> Channel 3/Output
//     PlcFastTask Outputs/.ARK_P1_050_DO02.PDOS.PlcToHw.digitalOutput_03 <-> Channel 4/Output
//     PlcFastTask Outputs/.ARK_P1_050_DO02.PDOS.PlcToHw.digitalOutput_04 <-> Channel 5/Output
//     PlcFastTask Outputs/.ARK_P1_050_DO02.PDOS.PlcToHw.digitalOutput_05 <-> Channel 6/Output
//     PlcFastTask Outputs/.ARK_P1_050_DO02.PDOS.PlcToHw.digitalOutput_06 <-> Channel 7/Output
//     PlcFastTask Outputs/.ARK_P1_050_DO02.PDOS.PlcToHw.digitalOutput_07 <-> Channel 8/Output
//     PlcFastTask Outputs/.ARK_P1_050_DO02.PDOS.PlcToHw.digitalOutput_08 <-> Channel 9/Output
//     PlcFastTask Outputs/.ARK_P1_050_DO02.PDOS.PlcToHw.digitalOutput_09 <-> Channel 10/Output
//     PlcFastTask Outputs/.ARK_P1_050_DO02.PDOS.PlcToHw.digitalOutput_10 <-> Channel 11/Output
//     PlcFastTask Outputs/.ARK_P1_050_DO02.PDOS.PlcToHw.digitalOutput_11 <-> Channel 12/Output
//     PlcFastTask Outputs/.ARK_P1_050_DO02.PDOS.PlcToHw.digitalOutput_12 <-> Channel 13/Output
//     PlcFastTask Outputs/.ARK_P1_050_DO02.PDOS.PlcToHw.digitalOutput_13 <-> Channel 14/Output
//     PlcFastTask Outputs/.ARK_P1_050_DO02.PDOS.PlcToHw.digitalOutput_14 <-> Channel 15/Output
//     PlcFastTask Outputs/.ARK_P1_050_DO02.PDOS.PlcToHw.digitalOutput_15 <-> Channel 16/Output
//   Plc_Program/Plc_Program Instance <-> ETC/SLT1+P1=050-BC1/SLT1+P1=050-DI1
//     PlcFastTask Inputs/.SLT1_P1_050_DI01.PDOS.digitalInput_00 <-> Channel 1/Input
//     PlcFastTask Inputs/.SLT1_P1_050_DI01.PDOS.digitalInput_01 <-> Channel 2/Input
//     PlcFastTask Inputs/.SLT1_P1_050_DI01.PDOS.digitalInput_02 <-> Channel 3/Input
//     PlcFastTask Inputs/.SLT1_P1_050_DI01.PDOS.digitalInput_03 <-> Channel 4/Input
//     PlcFastTask Inputs/.SLT1_P1_050_DI01.PDOS.digitalInput_04 <-> Channel 5/Input
//     PlcFastTask Inputs/.SLT1_P1_050_DI01.PDOS.digitalInput_05 <-> Channel 6/Input
//     PlcFastTask Inputs/.SLT1_P1_050_DI01.PDOS.digitalInput_06 <-> Channel 7/Input
//     PlcFastTask Inputs/.SLT1_P1_050_DI01.PDOS.digitalInput_07 <-> Channel 8/Input
//     PlcFastTask Inputs/.SLT1_P1_050_DI01.PDOS.digitalInput_08 <-> Channel 9/Input
//     PlcFastTask Inputs/.SLT1_P1_050_DI01.PDOS.digitalInput_09 <-> Channel 10/Input
//     PlcFastTask Inputs/.SLT1_P1_050_DI01.PDOS.digitalInput_10 <-> Channel 11/Input
//     PlcFastTask Inputs/.SLT1_P1_050_DI01.PDOS.digitalInput_11 <-> Channel 12/Input
//     PlcFastTask Inputs/.SLT1_P1_050_DI01.PDOS.digitalInput_12 <-> Channel 13/Input
//     PlcFastTask Inputs/.SLT1_P1_050_DI01.PDOS.digitalInput_13 <-> Channel 14/Input
//     PlcFastTask Inputs/.SLT1_P1_050_DI01.PDOS.digitalInput_14 <-> Channel 15/Input
//     PlcFastTask Inputs/.SLT1_P1_050_DI01.PDOS.digitalInput_15 <-> Channel 16/Input
//   Plc_Program/Plc_Program Instance <-> ETC/SLT1+P1=050-BC1/SLT1+P1=050-DI2
//     PlcFastTask Inputs/.SLT1_P1_050_DI02.PDOS.digitalInput_00 <-> Channel 1/Input
//     PlcFastTask Inputs/.SLT1_P1_050_DI02.PDOS.digitalInput_01 <-> Channel 2/Input
//     PlcFastTask Inputs/.SLT1_P1_050_DI02.PDOS.digitalInput_02 <-> Channel 3/Input
//     PlcFastTask Inputs/.SLT1_P1_050_DI02.PDOS.digitalInput_03 <-> Channel 4/Input
//     PlcFastTask Inputs/.SLT1_P1_050_DI02.PDOS.digitalInput_04 <-> Channel 5/Input
//     PlcFastTask Inputs/.SLT1_P1_050_DI02.PDOS.digitalInput_05 <-> Channel 6/Input
//     PlcFastTask Inputs/.SLT1_P1_050_DI02.PDOS.digitalInput_06 <-> Channel 7/Input
//     PlcFastTask Inputs/.SLT1_P1_050_DI02.PDOS.digitalInput_07 <-> Channel 8/Input
//     PlcFastTask Inputs/.SLT1_P1_050_DI02.PDOS.digitalInput_08 <-> Channel 9/Input
//     PlcFastTask Inputs/.SLT1_P1_050_DI02.PDOS.digitalInput_09 <-> Channel 10/Input
//     PlcFastTask Inputs/.SLT1_P1_050_DI02.PDOS.digitalInput_10 <-> Channel 11/Input
//     PlcFastTask Inputs/.SLT1_P1_050_DI02.PDOS.digitalInput_11 <-> Channel 12/Input
//     PlcFastTask Inputs/.SLT1_P1_050_DI02.PDOS.digitalInput_12 <-> Channel 13/Input
//     PlcFastTask Inputs/.SLT1_P1_050_DI02.PDOS.digitalInput_13 <-> Channel 14/Input
//     PlcFastTask Inputs/.SLT1_P1_050_DI02.PDOS.digitalInput_14 <-> Channel 15/Input
//     PlcFastTask Inputs/.SLT1_P1_050_DI02.PDOS.digitalInput_15 <-> Channel 16/Input
//   Plc_Program/Plc_Program Instance <-> ETC/SLT1+P1=050-BC1/SLT1+P1=050-DI3
//     PlcFastTask Inputs/.SLT1_P1_050_DI03.PDOS.digitalInput_00 <-> Channel 1/Input
//     PlcFastTask Inputs/.SLT1_P1_050_DI03.PDOS.digitalInput_01 <-> Channel 2/Input
//     PlcFastTask Inputs/.SLT1_P1_050_DI03.PDOS.digitalInput_02 <-> Channel 3/Input
//     PlcFastTask Inputs/.SLT1_P1_050_DI03.PDOS.digitalInput_03 <-> Channel 4/Input
//     PlcFastTask Inputs/.SLT1_P1_050_DI03.PDOS.digitalInput_04 <-> Channel 5/Input
//     PlcFastTask Inputs/.SLT1_P1_050_DI03.PDOS.digitalInput_05 <-> Channel 6/Input
//     PlcFastTask Inputs/.SLT1_P1_050_DI03.PDOS.digitalInput_06 <-> Channel 7/Input
//     PlcFastTask Inputs/.SLT1_P1_050_DI03.PDOS.digitalInput_07 <-> Channel 8/Input
//     PlcFastTask Inputs/.SLT1_P1_050_DI03.PDOS.digitalInput_08 <-> Channel 9/Input
//     PlcFastTask Inputs/.SLT1_P1_050_DI03.PDOS.digitalInput_09 <-> Channel 10/Input
//     PlcFastTask Inputs/.SLT1_P1_050_DI03.PDOS.digitalInput_10 <-> Channel 11/Input
//     PlcFastTask Inputs/.SLT1_P1_050_DI03.PDOS.digitalInput_11 <-> Channel 12/Input
//     PlcFastTask Inputs/.SLT1_P1_050_DI03.PDOS.digitalInput_12 <-> Channel 13/Input
//     PlcFastTask Inputs/.SLT1_P1_050_DI03.PDOS.digitalInput_13 <-> Channel 14/Input
//     PlcFastTask Inputs/.SLT1_P1_050_DI03.PDOS.digitalInput_14 <-> Channel 15/Input
//     PlcFastTask Inputs/.SLT1_P1_050_DI03.PDOS.digitalInput_15 <-> Channel 16/Input
//   Plc_Program/Plc_Program Instance <-> ETC/SLT1+P1=050-BC1/SLT1+P1=050-DI4
//     PlcFastTask Inputs/.SLT1_P1_050_DI04.PDOS.digitalInput_00 <-> Channel 1/Input
//     PlcFastTask Inputs/.SLT1_P1_050_DI04.PDOS.digitalInput_01 <-> Channel 2/Input
//     PlcFastTask Inputs/.SLT1_P1_050_DI04.PDOS.digitalInput_02 <-> Channel 3/Input
//     PlcFastTask Inputs/.SLT1_P1_050_DI04.PDOS.digitalInput_03 <-> Channel 4/Input
//     PlcFastTask Inputs/.SLT1_P1_050_DI04.PDOS.digitalInput_04 <-> Channel 5/Input
//     PlcFastTask Inputs/.SLT1_P1_050_DI04.PDOS.digitalInput_05 <-> Channel 6/Input
//     PlcFastTask Inputs/.SLT1_P1_050_DI04.PDOS.digitalInput_06 <-> Channel 7/Input
//     PlcFastTask Inputs/.SLT1_P1_050_DI04.PDOS.digitalInput_07 <-> Channel 8/Input
//     PlcFastTask Inputs/.SLT1_P1_050_DI04.PDOS.digitalInput_08 <-> Channel 9/Input
//     PlcFastTask Inputs/.SLT1_P1_050_DI04.PDOS.digitalInput_09 <-> Channel 10/Input
//     PlcFastTask Inputs/.SLT1_P1_050_DI04.PDOS.digitalInput_10 <-> Channel 11/Input
//     PlcFastTask Inputs/.SLT1_P1_050_DI04.PDOS.digitalInput_11 <-> Channel 12/Input
//     PlcFastTask Inputs/.SLT1_P1_050_DI04.PDOS.digitalInput_12 <-> Channel 13/Input
//     PlcFastTask Inputs/.SLT1_P1_050_DI04.PDOS.digitalInput_13 <-> Channel 14/Input
//     PlcFastTask Inputs/.SLT1_P1_050_DI04.PDOS.digitalInput_14 <-> Channel 15/Input
//     PlcFastTask Inputs/.SLT1_P1_050_DI04.PDOS.digitalInput_15 <-> Channel 16/Input
//   Plc_Program/Plc_Program Instance <-> ETC/SLT1+P1=050-BC1/SLT1+P1=050-DI5
//     PlcFastTask Inputs/.SLT1_P1_050_DI05.PDOS.digitalInput_00 <-> Channel 1/Input
//     PlcFastTask Inputs/.SLT1_P1_050_DI05.PDOS.digitalInput_01 <-> Channel 2/Input
//     PlcFastTask Inputs/.SLT1_P1_050_DI05.PDOS.digitalInput_02 <-> Channel 3/Input
//     PlcFastTask Inputs/.SLT1_P1_050_DI05.PDOS.digitalInput_03 <-> Channel 4/Input
//     PlcFastTask Inputs/.SLT1_P1_050_DI05.PDOS.digitalInput_04 <-> Channel 5/Input
//     PlcFastTask Inputs/.SLT1_P1_050_DI05.PDOS.digitalInput_05 <-> Channel 6/Input
//     PlcFastTask Inputs/.SLT1_P1_050_DI05.PDOS.digitalInput_06 <-> Channel 7/Input
//     PlcFastTask Inputs/.SLT1_P1_050_DI05.PDOS.digitalInput_07 <-> Channel 8/Input
//     PlcFastTask Inputs/.SLT1_P1_050_DI05.PDOS.digitalInput_08 <-> Channel 9/Input
//     PlcFastTask Inputs/.SLT1_P1_050_DI05.PDOS.digitalInput_09 <-> Channel 10/Input
//     PlcFastTask Inputs/.SLT1_P1_050_DI05.PDOS.digitalInput_10 <-> Channel 11/Input
//     PlcFastTask Inputs/.SLT1_P1_050_DI05.PDOS.digitalInput_11 <-> Channel 12/Input
//     PlcFastTask Inputs/.SLT1_P1_050_DI05.PDOS.digitalInput_12 <-> Channel 13/Input
//     PlcFastTask Inputs/.SLT1_P1_050_DI05.PDOS.digitalInput_13 <-> Channel 14/Input
//     PlcFastTask Inputs/.SLT1_P1_050_DI05.PDOS.digitalInput_14 <-> Channel 15/Input
//     PlcFastTask Inputs/.SLT1_P1_050_DI05.PDOS.digitalInput_15 <-> Channel 16/Input
//   Plc_Program/Plc_Program Instance <-> ETC/SLT1+P1=050-BC1/SLT1+P1=050-DO1
//     PlcFastTask Inputs/.SLT1_P1_050_DI06.PDOS.digitalInput_00 <-> Channel 1/Input
//     PlcFastTask Inputs/.SLT1_P1_050_DI06.PDOS.digitalInput_01 <-> Channel 2/Input
//     PlcFastTask Inputs/.SLT1_P1_050_DI06.PDOS.digitalInput_02 <-> Channel 3/Input
//     PlcFastTask Inputs/.SLT1_P1_050_DI06.PDOS.digitalInput_03 <-> Channel 4/Input
//     PlcFastTask Inputs/.SLT1_P1_050_DI06.PDOS.digitalInput_04 <-> Channel 5/Input
//     PlcFastTask Inputs/.SLT1_P1_050_DI06.PDOS.digitalInput_05 <-> Channel 6/Input
//     PlcFastTask Inputs/.SLT1_P1_050_DI06.PDOS.digitalInput_06 <-> Channel 7/Input
//     PlcFastTask Inputs/.SLT1_P1_050_DI06.PDOS.digitalInput_07 <-> Channel 8/Input
//     PlcFastTask Inputs/.SLT1_P1_050_DI06.PDOS.digitalInput_08 <-> Channel 9/Input
//     PlcFastTask Inputs/.SLT1_P1_050_DI06.PDOS.digitalInput_09 <-> Channel 10/Input
//     PlcFastTask Inputs/.SLT1_P1_050_DI06.PDOS.digitalInput_10 <-> Channel 11/Input
//     PlcFastTask Inputs/.SLT1_P1_050_DI06.PDOS.digitalInput_11 <-> Channel 12/Input
//     PlcFastTask Inputs/.SLT1_P1_050_DI06.PDOS.digitalInput_12 <-> Channel 13/Input
//     PlcFastTask Inputs/.SLT1_P1_050_DI06.PDOS.digitalInput_13 <-> Channel 14/Input
//     PlcFastTask Inputs/.SLT1_P1_050_DI06.PDOS.digitalInput_14 <-> Channel 15/Input
//     PlcFastTask Inputs/.SLT1_P1_050_DI06.PDOS.digitalInput_15 <-> Channel 16/Input
//   Plc_Program/Plc_Program Instance <-> ETC/SLT1+P1=050-BC1/SLT1+P1=050-DO2
//     PlcFastTask Outputs/.SLT1_P1_050_DO01.PDOS.PlcToHw.digitalOutput_00 <-> Channel 1/Output
//     PlcFastTask Outputs/.SLT1_P1_050_DO01.PDOS.PlcToHw.digitalOutput_01 <-> Channel 2/Output
//     PlcFastTask Outputs/.SLT1_P1_050_DO01.PDOS.PlcToHw.digitalOutput_02 <-> Channel 3/Output
//     PlcFastTask Outputs/.SLT1_P1_050_DO01.PDOS.PlcToHw.digitalOutput_03 <-> Channel 4/Output
//     PlcFastTask Outputs/.SLT1_P1_050_DO01.PDOS.PlcToHw.digitalOutput_04 <-> Channel 5/Output
//     PlcFastTask Outputs/.SLT1_P1_050_DO01.PDOS.PlcToHw.digitalOutput_05 <-> Channel 6/Output
//     PlcFastTask Outputs/.SLT1_P1_050_DO01.PDOS.PlcToHw.digitalOutput_06 <-> Channel 7/Output
//     PlcFastTask Outputs/.SLT1_P1_050_DO01.PDOS.PlcToHw.digitalOutput_07 <-> Channel 8/Output
//     PlcFastTask Outputs/.SLT1_P1_050_DO01.PDOS.PlcToHw.digitalOutput_08 <-> Channel 9/Output
//     PlcFastTask Outputs/.SLT1_P1_050_DO01.PDOS.PlcToHw.digitalOutput_09 <-> Channel 10/Output
//     PlcFastTask Outputs/.SLT1_P1_050_DO01.PDOS.PlcToHw.digitalOutput_10 <-> Channel 11/Output
//     PlcFastTask Outputs/.SLT1_P1_050_DO01.PDOS.PlcToHw.digitalOutput_11 <-> Channel 12/Output
//     PlcFastTask Outputs/.SLT1_P1_050_DO01.PDOS.PlcToHw.digitalOutput_12 <-> Channel 13/Output
//     PlcFastTask Outputs/.SLT1_P1_050_DO01.PDOS.PlcToHw.digitalOutput_13 <-> Channel 14/Output
//     PlcFastTask Outputs/.SLT1_P1_050_DO01.PDOS.PlcToHw.digitalOutput_14 <-> Channel 15/Output
//     PlcFastTask Outputs/.SLT1_P1_050_DO01.PDOS.PlcToHw.digitalOutput_15 <-> Channel 16/Output
//   Plc_Program/Plc_Program Instance <-> ETC/SLT1+P1=050-BC1/SLT1+P1=050-DO3
//     PlcFastTask Outputs/.SLT1_P1_050_DO02.PDOS.PlcToHw.digitalOutput_00 <-> Channel 1/Output
//     PlcFastTask Outputs/.SLT1_P1_050_DO02.PDOS.PlcToHw.digitalOutput_01 <-> Channel 2/Output
//     PlcFastTask Outputs/.SLT1_P1_050_DO02.PDOS.PlcToHw.digitalOutput_02 <-> Channel 3/Output
//     PlcFastTask Outputs/.SLT1_P1_050_DO02.PDOS.PlcToHw.digitalOutput_03 <-> Channel 4/Output
//     PlcFastTask Outputs/.SLT1_P1_050_DO02.PDOS.PlcToHw.digitalOutput_04 <-> Channel 5/Output
//     PlcFastTask Outputs/.SLT1_P1_050_DO02.PDOS.PlcToHw.digitalOutput_05 <-> Channel 6/Output
//     PlcFastTask Outputs/.SLT1_P1_050_DO02.PDOS.PlcToHw.digitalOutput_06 <-> Channel 7/Output
//     PlcFastTask Outputs/.SLT1_P1_050_DO02.PDOS.PlcToHw.digitalOutput_07 <-> Channel 8/Output
//     PlcFastTask Outputs/.SLT1_P1_050_DO02.PDOS.PlcToHw.digitalOutput_08 <-> Channel 9/Output
//     PlcFastTask Outputs/.SLT1_P1_050_DO02.PDOS.PlcToHw.digitalOutput_09 <-> Channel 10/Output
//     PlcFastTask Outputs/.SLT1_P1_050_DO02.PDOS.PlcToHw.digitalOutput_10 <-> Channel 11/Output
//     PlcFastTask Outputs/.SLT1_P1_050_DO02.PDOS.PlcToHw.digitalOutput_11 <-> Channel 12/Output
//     PlcFastTask Outputs/.SLT1_P1_050_DO02.PDOS.PlcToHw.digitalOutput_12 <-> Channel 13/Output
//     PlcFastTask Outputs/.SLT1_P1_050_DO02.PDOS.PlcToHw.digitalOutput_13 <-> Channel 14/Output
//     PlcFastTask Outputs/.SLT1_P1_050_DO02.PDOS.PlcToHw.digitalOutput_14 <-> Channel 15/Output
//     PlcFastTask Outputs/.SLT1_P1_050_DO02.PDOS.PlcToHw.digitalOutput_15 <-> Channel 16/Output
//   Plc_Program/Plc_Program Instance <-> ETC/SLT1+P1=050-BC1/SLT1+P1=050-DO4
//     PlcFastTask Outputs/.SLT1_P1_050_DO03.PDOS.PlcToHw.digitalOutput_00 <-> Channel 1/Output
//     PlcFastTask Outputs/.SLT1_P1_050_DO03.PDOS.PlcToHw.digitalOutput_01 <-> Channel 2/Output
//     PlcFastTask Outputs/.SLT1_P1_050_DO03.PDOS.PlcToHw.digitalOutput_02 <-> Channel 3/Output
//     PlcFastTask Outputs/.SLT1_P1_050_DO03.PDOS.PlcToHw.digitalOutput_03 <-> Channel 4/Output
//     PlcFastTask Outputs/.SLT1_P1_050_DO03.PDOS.PlcToHw.digitalOutput_04 <-> Channel 5/Output
//     PlcFastTask Outputs/.SLT1_P1_050_DO03.PDOS.PlcToHw.digitalOutput_05 <-> Channel 6/Output
//     PlcFastTask Outputs/.SLT1_P1_050_DO03.PDOS.PlcToHw.digitalOutput_06 <-> Channel 7/Output
//     PlcFastTask Outputs/.SLT1_P1_050_DO03.PDOS.PlcToHw.digitalOutput_07 <-> Channel 8/Output
//     PlcFastTask Outputs/.SLT1_P1_050_DO03.PDOS.PlcToHw.digitalOutput_08 <-> Channel 9/Output
//     PlcFastTask Outputs/.SLT1_P1_050_DO03.PDOS.PlcToHw.digitalOutput_09 <-> Channel 10/Output
//     PlcFastTask Outputs/.SLT1_P1_050_DO03.PDOS.PlcToHw.digitalOutput_10 <-> Channel 11/Output
//     PlcFastTask Outputs/.SLT1_P1_050_DO03.PDOS.PlcToHw.digitalOutput_11 <-> Channel 12/Output
//     PlcFastTask Outputs/.SLT1_P1_050_DO03.PDOS.PlcToHw.digitalOutput_12 <-> Channel 13/Output
//     PlcFastTask Outputs/.SLT1_P1_050_DO03.PDOS.PlcToHw.digitalOutput_13 <-> Channel 14/Output
//     PlcFastTask Outputs/.SLT1_P1_050_DO03.PDOS.PlcToHw.digitalOutput_14 <-> Channel 15/Output
//     PlcFastTask Outputs/.SLT1_P1_050_DO03.PDOS.PlcToHw.digitalOutput_15 <-> Channel 16/Output
//   Plc_Program/Plc_Program Instance <-> ETC/SLT1+P1=050-BC1/SLT1+P1=050-DO5
//     PlcFastTask Outputs/.SLT1_P1_050_DO04.PDOS.PlcToHw.digitalOutput_00 <-> Channel 1/Output
//     PlcFastTask Outputs/.SLT1_P1_050_DO04.PDOS.PlcToHw.digitalOutput_01 <-> Channel 2/Output
//     PlcFastTask Outputs/.SLT1_P1_050_DO04.PDOS.PlcToHw.digitalOutput_02 <-> Channel 3/Output
//     PlcFastTask Outputs/.SLT1_P1_050_DO04.PDOS.PlcToHw.digitalOutput_03 <-> Channel 4/Output
//     PlcFastTask Outputs/.SLT1_P1_050_DO04.PDOS.PlcToHw.digitalOutput_04 <-> Channel 5/Output
//     PlcFastTask Outputs/.SLT1_P1_050_DO04.PDOS.PlcToHw.digitalOutput_05 <-> Channel 6/Output
//     PlcFastTask Outputs/.SLT1_P1_050_DO04.PDOS.PlcToHw.digitalOutput_06 <-> Channel 7/Output
//     PlcFastTask Outputs/.SLT1_P1_050_DO04.PDOS.PlcToHw.digitalOutput_07 <-> Channel 8/Output
//     PlcFastTask Outputs/.SLT1_P1_050_DO04.PDOS.PlcToHw.digitalOutput_08 <-> Channel 9/Output
//     PlcFastTask Outputs/.SLT1_P1_050_DO04.PDOS.PlcToHw.digitalOutput_09 <-> Channel 10/Output
//     PlcFastTask Outputs/.SLT1_P1_050_DO04.PDOS.PlcToHw.digitalOutput_10 <-> Channel 11/Output
//     PlcFastTask Outputs/.SLT1_P1_050_DO04.PDOS.PlcToHw.digitalOutput_11 <-> Channel 12/Output
//     PlcFastTask Outputs/.SLT1_P1_050_DO04.PDOS.PlcToHw.digitalOutput_12 <-> Channel 13/Output
//     PlcFastTask Outputs/.SLT1_P1_050_DO04.PDOS.PlcToHw.digitalOutput_13 <-> Channel 14/Output
//     PlcFastTask Outputs/.SLT1_P1_050_DO04.PDOS.PlcToHw.digitalOutput_14 <-> Channel 15/Output
//     PlcFastTask Outputs/.SLT1_P1_050_DO04.PDOS.PlcToHw.digitalOutput_15 <-> Channel 16/Output
//   Plc_Program/Plc_Program Instance <-> ETC/SLT1+P1=050-BC1/SLT1+P1=050-DO6
//     PlcFastTask Outputs/.SLT1_P1_050_DO05.PDOS.PlcToHw.digitalOutput_00 <-> Channel 1/Output
//     PlcFastTask Outputs/.SLT1_P1_050_DO05.PDOS.PlcToHw.digitalOutput_01 <-> Channel 2/Output
//     PlcFastTask Outputs/.SLT1_P1_050_DO05.PDOS.PlcToHw.digitalOutput_02 <-> Channel 3/Output
//     PlcFastTask Outputs/.SLT1_P1_050_DO05.PDOS.PlcToHw.digitalOutput_03 <-> Channel 4/Output
//     PlcFastTask Outputs/.SLT1_P1_050_DO05.PDOS.PlcToHw.digitalOutput_04 <-> Channel 5/Output
//     PlcFastTask Outputs/.SLT1_P1_050_DO05.PDOS.PlcToHw.digitalOutput_05 <-> Channel 6/Output
//     PlcFastTask Outputs/.SLT1_P1_050_DO05.PDOS.PlcToHw.digitalOutput_06 <-> Channel 7/Output
//     PlcFastTask Outputs/.SLT1_P1_050_DO05.PDOS.PlcToHw.digitalOutput_07 <-> Channel 8/Output
//     PlcFastTask Outputs/.SLT1_P1_050_DO05.PDOS.PlcToHw.digitalOutput_08 <-> Channel 9/Output
//     PlcFastTask Outputs/.SLT1_P1_050_DO05.PDOS.PlcToHw.digitalOutput_09 <-> Channel 10/Output
//     PlcFastTask Outputs/.SLT1_P1_050_DO05.PDOS.PlcToHw.digitalOutput_10 <-> Channel 11/Output
//     PlcFastTask Outputs/.SLT1_P1_050_DO05.PDOS.PlcToHw.digitalOutput_11 <-> Channel 12/Output
//     PlcFastTask Outputs/.SLT1_P1_050_DO05.PDOS.PlcToHw.digitalOutput_12 <-> Channel 13/Output
//     PlcFastTask Outputs/.SLT1_P1_050_DO05.PDOS.PlcToHw.digitalOutput_13 <-> Channel 14/Output
//     PlcFastTask Outputs/.SLT1_P1_050_DO05.PDOS.PlcToHw.digitalOutput_14 <-> Channel 15/Output
//     PlcFastTask Outputs/.SLT1_P1_050_DO05.PDOS.PlcToHw.digitalOutput_15 <-> Channel 16/Output
//   Plc_Program/Plc_Program Instance <-> ETC/SLT1+P1=050-BC1/SLT1+P1=050-DO7
//     PlcFastTask Outputs/.SLT1_P1_050_DO06.PDOS.PlcToHw.digitalOutput_00 <-> Channel 1/Output
//     PlcFastTask Outputs/.SLT1_P1_050_DO06.PDOS.PlcToHw.digitalOutput_01 <-> Channel 2/Output
//     PlcFastTask Outputs/.SLT1_P1_050_DO06.PDOS.PlcToHw.digitalOutput_02 <-> Channel 3/Output
//     PlcFastTask Outputs/.SLT1_P1_050_DO06.PDOS.PlcToHw.digitalOutput_03 <-> Channel 4/Output
//     PlcFastTask Outputs/.SLT1_P1_050_DO06.PDOS.PlcToHw.digitalOutput_04 <-> Channel 5/Output
//     PlcFastTask Outputs/.SLT1_P1_050_DO06.PDOS.PlcToHw.digitalOutput_05 <-> Channel 6/Output
//     PlcFastTask Outputs/.SLT1_P1_050_DO06.PDOS.PlcToHw.digitalOutput_06 <-> Channel 7/Output
//     PlcFastTask Outputs/.SLT1_P1_050_DO06.PDOS.PlcToHw.digitalOutput_07 <-> Channel 8/Output
//     PlcFastTask Outputs/.SLT1_P1_050_DO06.PDOS.PlcToHw.digitalOutput_08 <-> Channel 9/Output
//     PlcFastTask Outputs/.SLT1_P1_050_DO06.PDOS.PlcToHw.digitalOutput_09 <-> Channel 10/Output
//     PlcFastTask Outputs/.SLT1_P1_050_DO06.PDOS.PlcToHw.digitalOutput_10 <-> Channel 11/Output
//     PlcFastTask Outputs/.SLT1_P1_050_DO06.PDOS.PlcToHw.digitalOutput_11 <-> Channel 12/Output
//     PlcFastTask Outputs/.SLT1_P1_050_DO06.PDOS.PlcToHw.digitalOutput_12 <-> Channel 13/Output
//     PlcFastTask Outputs/.SLT1_P1_050_DO06.PDOS.PlcToHw.digitalOutput_13 <-> Channel 14/Output
//     PlcFastTask Outputs/.SLT1_P1_050_DO06.PDOS.PlcToHw.digitalOutput_14 <-> Channel 15/Output
//     PlcFastTask Outputs/.SLT1_P1_050_DO06.PDOS.PlcToHw.digitalOutput_15 <-> Channel 16/Output
//   Plc_Program/Plc_Program Instance <-> ETC/STK+M=050-BC1
//     PlcTask Inputs/.STKL_050_DIO1.HwToPlc/inputByte_0 <-> STKL+M=050-DIO1 - IO-Link slave IP67 [Machine drive side]/IO-Link Input process data mapping/Input Byte 0
//     PlcTask Inputs/.STKL_050_DIO1.HwToPlc/inputByte_1 <-> STKL+M=050-DIO1 - IO-Link slave IP67 [Machine drive side]/IO-Link Input process data mapping/Input Byte 1
//     PlcTask Inputs/.STKL_050_DIO2.HwToPlc/inputByte_0 <-> STKL+M=050-DIO2  - IO-Link slave IP24 [Lower command box]/IO-Link Input process data mapping/Input Byte 0
//     PlcTask Inputs/.STKL_050_DIO2.HwToPlc/inputByte_1 <-> STKL+M=050-DIO2  - IO-Link slave IP24 [Lower command box]/IO-Link Input process data mapping/Input Byte 1
//     PlcTask Inputs/.STKL_100_B01.HwToPlc/inputByte_0 <-> STKL+M=050-BE1  - IO-Link Sick distance sensor [Backstop]/IO-Link Input process data mapping/Input Byte 0
//     PlcTask Inputs/.STKL_100_B01.HwToPlc/inputByte_1 <-> STKL+M=050-BE1  - IO-Link Sick distance sensor [Backstop]/IO-Link Input process data mapping/Input Byte 1
//     PlcTask Inputs/.STKU_050_DIO1.HwToPlc/inputByte_0 <-> STKU+M=050-DIO1  - IO-Link slave IP24 [Lower command box]/IO-Link Input process data mapping/Input Byte 0
//     PlcTask Inputs/.STKU_050_DIO1.HwToPlc/inputByte_1 <-> STKU+M=050-DIO1  - IO-Link slave IP24 [Lower command box]/IO-Link Input process data mapping/Input Byte 1
//     PlcTask Inputs/.STKU_050_DIO2.HwToPlc/inputByte_0 <-> STKU+M=050-DIO2  - IO-Link slave IP24 [Uppercommand box]/IO-Link Input process data mapping/Input Byte 0
//     PlcTask Inputs/.STKU_050_DIO2.HwToPlc/inputByte_1 <-> STKU+M=050-DIO2  - IO-Link slave IP24 [Uppercommand box]/IO-Link Input process data mapping/Input Byte 1
//     PlcTask Inputs/.STKU_050_DIO3.HwToPlc/inputByte_0 <-> STKU+M=050-DIO3  - IO-Link slave IP24 [Elevator drive side]/IO-Link Input process data mapping/Input Byte 0
//     PlcTask Inputs/.STKU_050_DIO3.HwToPlc/inputByte_1 <-> STKU+M=050-DIO3  - IO-Link slave IP24 [Elevator drive side]/IO-Link Input process data mapping/Input Byte 1
//     PlcTask Inputs/.STK_050_BC2.HwToPlc/deviceState <-> Digital Input Mapping/Device Status
//     PlcTask Inputs/.STK_050_BC2.HwToPlc/inputPin2 <-> Digital Input Mapping/Actuator Shutdown Pin 2
//     PlcTask Inputs/.STK_050_BC2.HwToPlc/inputPin4 <-> Digital Input Mapping/Input Pin 4
//     PlcTask Inputs/.STK_050_BC2.HwToPlc/ioLinkDeviceState_Port0 <-> IO-Link Device State/Status Of IO-Link Port 0
//     PlcTask Inputs/.STK_050_BC2.HwToPlc/ioLinkDeviceState_Port1 <-> IO-Link Device State/Status Of IO-Link Port 1
//     PlcTask Inputs/.STK_050_BC2.HwToPlc/ioLinkDeviceState_Port2 <-> IO-Link Device State/Status Of IO-Link Port 2
//     PlcTask Inputs/.STK_050_BC2.HwToPlc/ioLinkDeviceState_Port3 <-> IO-Link Device State/Status Of IO-Link Port 3
//     PlcTask Inputs/.STK_050_BC2.HwToPlc/ioLinkDeviceState_Port4 <-> IO-Link Device State/Status Of IO-Link Port 4
//     PlcTask Inputs/.STK_050_BC2.HwToPlc/ioLinkDeviceState_Port5 <-> IO-Link Device State/Status Of IO-Link Port 5
//     PlcTask Inputs/.STK_050_BC2.HwToPlc/ioLinkDeviceState_Port6 <-> IO-Link Device State/Status Of IO-Link Port 6
//     PlcTask Inputs/.STK_050_BC2.HwToPlc/ioLinkDeviceState_Port7 <-> IO-Link Device State/Status Of IO-Link Port 7
//     PlcTask Outputs/.STKL_050_DIO1.PlcToHw/outputByte_0 <-> STKL+M=050-DIO1 - IO-Link slave IP67 [Machine drive side]/IO-Link Output process data mapping/Output Byte 0
//     PlcTask Outputs/.STKL_050_DIO1.PlcToHw/outputByte_1 <-> STKL+M=050-DIO1 - IO-Link slave IP67 [Machine drive side]/IO-Link Output process data mapping/Output Byte 1
//     PlcTask Outputs/.STKL_050_DIO2.PlcToHw/outputByte_0 <-> STKL+M=050-DIO2  - IO-Link slave IP24 [Lower command box]/IO-Link Output process data mapping/Output Byte 0
//     PlcTask Outputs/.STKL_050_DIO2.PlcToHw/outputByte_1 <-> STKL+M=050-DIO2  - IO-Link slave IP24 [Lower command box]/IO-Link Output process data mapping/Output Byte 1
//     PlcTask Outputs/.STKU_050_DIO1.PlcToHw/outputByte_0 <-> STKU+M=050-DIO1  - IO-Link slave IP24 [Lower command box]/IO-Link Output process data mapping/Output Byte 0
//     PlcTask Outputs/.STKU_050_DIO1.PlcToHw/outputByte_1 <-> STKU+M=050-DIO1  - IO-Link slave IP24 [Lower command box]/IO-Link Output process data mapping/Output Byte 1
//     PlcTask Outputs/.STKU_050_DIO2.PlcToHw/outputByte_0 <-> STKU+M=050-DIO2  - IO-Link slave IP24 [Uppercommand box]/IO-Link Output process data mapping/Output Byte 0
//     PlcTask Outputs/.STKU_050_DIO2.PlcToHw/outputByte_1 <-> STKU+M=050-DIO2  - IO-Link slave IP24 [Uppercommand box]/IO-Link Output process data mapping/Output Byte 1
//     PlcTask Outputs/.STKU_050_DIO3.PlcToHw/outputByte_0 <-> STKU+M=050-DIO3  - IO-Link slave IP24 [Elevator drive side]/IO-Link Output process data mapping/Output Byte 0
//     PlcTask Outputs/.STKU_050_DIO3.PlcToHw/outputByte_1 <-> STKU+M=050-DIO3  - IO-Link slave IP24 [Elevator drive side]/IO-Link Output process data mapping/Output Byte 1
//   Plc_Program/Plc_Program Instance <-> ETC/STK+P2=050-BC1/STK+P2=050-AO1
//     PlcTask Outputs/.STK_P2_050_AO1.PDOS.HwToPLC.Channel1 <-> AO Outputs Channel 1/Analog output
//     PlcTask Outputs/.STK_P2_050_AO1.PDOS.HwToPLC.Channel2 <-> AO Outputs Channel 2/Analog output
//     PlcTask Outputs/.STK_P2_050_AO1.PDOS.HwToPLC.Channel3 <-> AO Outputs Channel 3/Analog output
//     PlcTask Outputs/.STK_P2_050_AO1.PDOS.HwToPLC.Channel4 <-> AO Outputs Channel 4/Analog output
//   Plc_Program/Plc_Program Instance <-> ETC/STK+P2=050-BC1/STK+P2=050-AO2
//     PlcTask Outputs/.STK_P2_050_AO2.PDOS.HwToPLC.Channel1 <-> AO Outputs Channel 1/Analog output
//     PlcTask Outputs/.STK_P2_050_AO2.PDOS.HwToPLC.Channel2 <-> AO Outputs Channel 2/Analog output
//     PlcTask Outputs/.STK_P2_050_AO2.PDOS.HwToPLC.Channel3 <-> AO Outputs Channel 3/Analog output
//     PlcTask Outputs/.STK_P2_050_AO2.PDOS.HwToPLC.Channel4 <-> AO Outputs Channel 4/Analog output
//   Plc_Program/Plc_Program Instance <-> ETC/STK+P2=050-BC1/STK+P2=050-AO3
//     PlcTask Outputs/.STK_P2_050_AO3.PDOS.HwToPLC.Channel1 <-> AO Outputs Channel 1/Analog output
//     PlcTask Outputs/.STK_P2_050_AO3.PDOS.HwToPLC.Channel2 <-> AO Outputs Channel 2/Analog output
//     PlcTask Outputs/.STK_P2_050_AO3.PDOS.HwToPLC.Channel3 <-> AO Outputs Channel 3/Analog output
//     PlcTask Outputs/.STK_P2_050_AO3.PDOS.HwToPLC.Channel4 <-> AO Outputs Channel 4/Analog output
//   Plc_Program/Plc_Program Instance <-> ETC/STK+P2=050-BC1/STK+P2=050-AO4
//     PlcTask Outputs/.STK_P2_050_AO4.PDOS.HwToPLC.Channel1 <-> AO Outputs Channel 1/Analog output
//     PlcTask Outputs/.STK_P2_050_AO4.PDOS.HwToPLC.Channel2 <-> AO Outputs Channel 2/Analog output
//     PlcTask Outputs/.STK_P2_050_AO4.PDOS.HwToPLC.Channel3 <-> AO Outputs Channel 3/Analog output
//     PlcTask Outputs/.STK_P2_050_AO4.PDOS.HwToPLC.Channel4 <-> AO Outputs Channel 4/Analog output
//   Plc_Program/Plc_Program Instance <-> ETC/STK+P2=050-BC1/STK+P2=050-DI1
//     PlcTask Inputs/.STK_P2_050_DI1.PDOS.digitalInput_00 <-> Channel 1/Input
//     PlcTask Inputs/.STK_P2_050_DI1.PDOS.digitalInput_01 <-> Channel 2/Input
//     PlcTask Inputs/.STK_P2_050_DI1.PDOS.digitalInput_02 <-> Channel 3/Input
//     PlcTask Inputs/.STK_P2_050_DI1.PDOS.digitalInput_03 <-> Channel 4/Input
//     PlcTask Inputs/.STK_P2_050_DI1.PDOS.digitalInput_04 <-> Channel 5/Input
//     PlcTask Inputs/.STK_P2_050_DI1.PDOS.digitalInput_05 <-> Channel 6/Input
//     PlcTask Inputs/.STK_P2_050_DI1.PDOS.digitalInput_06 <-> Channel 7/Input
//     PlcTask Inputs/.STK_P2_050_DI1.PDOS.digitalInput_07 <-> Channel 8/Input
//     PlcTask Inputs/.STK_P2_050_DI1.PDOS.digitalInput_08 <-> Channel 9/Input
//     PlcTask Inputs/.STK_P2_050_DI1.PDOS.digitalInput_09 <-> Channel 10/Input
//     PlcTask Inputs/.STK_P2_050_DI1.PDOS.digitalInput_10 <-> Channel 11/Input
//     PlcTask Inputs/.STK_P2_050_DI1.PDOS.digitalInput_11 <-> Channel 12/Input
//     PlcTask Inputs/.STK_P2_050_DI1.PDOS.digitalInput_12 <-> Channel 13/Input
//     PlcTask Inputs/.STK_P2_050_DI1.PDOS.digitalInput_13 <-> Channel 14/Input
//     PlcTask Inputs/.STK_P2_050_DI1.PDOS.digitalInput_14 <-> Channel 15/Input
//     PlcTask Inputs/.STK_P2_050_DI1.PDOS.digitalInput_15 <-> Channel 16/Input
//   Plc_Program/Plc_Program Instance <-> ETC/STK+P2=050-BC1/STK+P2=050-DI2
//     PlcTask Inputs/.STK_P2_050_DI2.PDOS.digitalInput_00 <-> Channel 1/Input
//     PlcTask Inputs/.STK_P2_050_DI2.PDOS.digitalInput_01 <-> Channel 2/Input
//     PlcTask Inputs/.STK_P2_050_DI2.PDOS.digitalInput_02 <-> Channel 3/Input
//     PlcTask Inputs/.STK_P2_050_DI2.PDOS.digitalInput_03 <-> Channel 4/Input
//     PlcTask Inputs/.STK_P2_050_DI2.PDOS.digitalInput_04 <-> Channel 5/Input
//     PlcTask Inputs/.STK_P2_050_DI2.PDOS.digitalInput_05 <-> Channel 6/Input
//     PlcTask Inputs/.STK_P2_050_DI2.PDOS.digitalInput_06 <-> Channel 7/Input
//     PlcTask Inputs/.STK_P2_050_DI2.PDOS.digitalInput_07 <-> Channel 8/Input
//     PlcTask Inputs/.STK_P2_050_DI2.PDOS.digitalInput_08 <-> Channel 9/Input
//     PlcTask Inputs/.STK_P2_050_DI2.PDOS.digitalInput_09 <-> Channel 10/Input
//     PlcTask Inputs/.STK_P2_050_DI2.PDOS.digitalInput_10 <-> Channel 11/Input
//     PlcTask Inputs/.STK_P2_050_DI2.PDOS.digitalInput_11 <-> Channel 12/Input
//     PlcTask Inputs/.STK_P2_050_DI2.PDOS.digitalInput_12 <-> Channel 13/Input
//     PlcTask Inputs/.STK_P2_050_DI2.PDOS.digitalInput_13 <-> Channel 14/Input
//     PlcTask Inputs/.STK_P2_050_DI2.PDOS.digitalInput_14 <-> Channel 15/Input
//     PlcTask Inputs/.STK_P2_050_DI2.PDOS.digitalInput_15 <-> Channel 16/Input
//   Plc_Program/Plc_Program Instance <-> ETC/STK+P2=050-BC1/STK+P2=050-DO1
//     PlcTask Outputs/.STK_P2_050_DO1.PDOS.PlcToHw.digitalOutput_00 <-> Channel 1/Output
//     PlcTask Outputs/.STK_P2_050_DO1.PDOS.PlcToHw.digitalOutput_01 <-> Channel 2/Output
//     PlcTask Outputs/.STK_P2_050_DO1.PDOS.PlcToHw.digitalOutput_02 <-> Channel 3/Output
//     PlcTask Outputs/.STK_P2_050_DO1.PDOS.PlcToHw.digitalOutput_03 <-> Channel 4/Output
//     PlcTask Outputs/.STK_P2_050_DO1.PDOS.PlcToHw.digitalOutput_04 <-> Channel 5/Output
//     PlcTask Outputs/.STK_P2_050_DO1.PDOS.PlcToHw.digitalOutput_05 <-> Channel 6/Output
//     PlcTask Outputs/.STK_P2_050_DO1.PDOS.PlcToHw.digitalOutput_06 <-> Channel 7/Output
//     PlcTask Outputs/.STK_P2_050_DO1.PDOS.PlcToHw.digitalOutput_07 <-> Channel 8/Output
//     PlcTask Outputs/.STK_P2_050_DO1.PDOS.PlcToHw.digitalOutput_08 <-> Channel 9/Output
//     PlcTask Outputs/.STK_P2_050_DO1.PDOS.PlcToHw.digitalOutput_09 <-> Channel 10/Output
//     PlcTask Outputs/.STK_P2_050_DO1.PDOS.PlcToHw.digitalOutput_10 <-> Channel 11/Output
//     PlcTask Outputs/.STK_P2_050_DO1.PDOS.PlcToHw.digitalOutput_11 <-> Channel 12/Output
//     PlcTask Outputs/.STK_P2_050_DO1.PDOS.PlcToHw.digitalOutput_12 <-> Channel 13/Output
//     PlcTask Outputs/.STK_P2_050_DO1.PDOS.PlcToHw.digitalOutput_13 <-> Channel 14/Output
//     PlcTask Outputs/.STK_P2_050_DO1.PDOS.PlcToHw.digitalOutput_14 <-> Channel 15/Output
//     PlcTask Outputs/.STK_P2_050_DO1.PDOS.PlcToHw.digitalOutput_15 <-> Channel 16/Output
//   Plc_Program/Plc_Program Instance <-> ETC/STK+P2=050-BC1/STK+P2=050-DO2
//     PlcTask Outputs/.STK_P2_050_DO2.PDOS.PlcToHw.digitalOutput_00 <-> Channel 1/Output
//     PlcTask Outputs/.STK_P2_050_DO2.PDOS.PlcToHw.digitalOutput_01 <-> Channel 2/Output
//     PlcTask Outputs/.STK_P2_050_DO2.PDOS.PlcToHw.digitalOutput_02 <-> Channel 3/Output
//     PlcTask Outputs/.STK_P2_050_DO2.PDOS.PlcToHw.digitalOutput_03 <-> Channel 4/Output
//     PlcTask Outputs/.STK_P2_050_DO2.PDOS.PlcToHw.digitalOutput_04 <-> Channel 5/Output
//     PlcTask Outputs/.STK_P2_050_DO2.PDOS.PlcToHw.digitalOutput_05 <-> Channel 6/Output
//     PlcTask Outputs/.STK_P2_050_DO2.PDOS.PlcToHw.digitalOutput_06 <-> Channel 7/Output
//     PlcTask Outputs/.STK_P2_050_DO2.PDOS.PlcToHw.digitalOutput_07 <-> Channel 8/Output
//     PlcTask Outputs/.STK_P2_050_DO2.PDOS.PlcToHw.digitalOutput_08 <-> Channel 9/Output
//     PlcTask Outputs/.STK_P2_050_DO2.PDOS.PlcToHw.digitalOutput_09 <-> Channel 10/Output
//     PlcTask Outputs/.STK_P2_050_DO2.PDOS.PlcToHw.digitalOutput_10 <-> Channel 11/Output
//     PlcTask Outputs/.STK_P2_050_DO2.PDOS.PlcToHw.digitalOutput_11 <-> Channel 12/Output
//     PlcTask Outputs/.STK_P2_050_DO2.PDOS.PlcToHw.digitalOutput_12 <-> Channel 13/Output
//     PlcTask Outputs/.STK_P2_050_DO2.PDOS.PlcToHw.digitalOutput_13 <-> Channel 14/Output
//     PlcTask Outputs/.STK_P2_050_DO2.PDOS.PlcToHw.digitalOutput_14 <-> Channel 15/Output
//     PlcTask Outputs/.STK_P2_050_DO2.PDOS.PlcToHw.digitalOutput_15 <-> Channel 16/Output
//   Plc_Program/Plc_Program Instance <-> ETC/STK+P2=050-BC1/STK+P2=050-ENC1
//     PlcTask Inputs/.STK_P2_050_ENC1.HwToPlc/channel1/CounterValue <-> ENC Status Channel 1/Counter value
//     PlcTask Inputs/.STK_P2_050_ENC1.HwToPlc/channel2/CounterValue <-> ENC Status Channel 2/Counter value
//     PlcTask Inputs/.STK_P2_050_ENC1.HwToPlc/channel1/status <-> ENC Status Channel 1/Status
//     PlcTask Inputs/.STK_P2_050_ENC1.HwToPlc/channel2/status <-> ENC Status Channel 2/Status
//     PlcTask Outputs/.STK_P2_050_ENC1.PlcToHw/channel1/control/Set_counter <-> ENC Control Channel 1/Control/Set counter
//     PlcTask Outputs/.STK_P2_050_ENC1.PlcToHw/channel2/control/Set_counter <-> ENC Control Channel 2/Control/Set counter
//     PlcTask Outputs/.STK_P2_050_ENC1.PlcToHw/channel1/setCounterValue <-> ENC Control Channel 1/Set counter value
//     PlcTask Outputs/.STK_P2_050_ENC1.PlcToHw/channel2/setCounterValue <-> ENC Control Channel 2/Set counter value
//   Plc_Program/Plc_Program Instance <-> ETC/STK+P2=050-BC1/STK+P2=050-SP1
//     PlcTask Inputs/.STK_P2_050_SP01.PDOS.HwToPLC.EStop1Diag <-> Function Block Info Data/TwinSafeGroup1.Network1.FBEstop2 Info Data/Diag
//     PlcTask Inputs/.STK_P2_050_SP01.PDOS.HwToPLC.EStop2Diag <-> Function Block Info Data/TwinSafeGroup1.Network1.FBEstop1 Info Data/Diag
//     PlcTask Inputs/.STK_P2_050_SP01.PDOS.HwToPLC.EStop1State <-> Function Block Info Data/TwinSafeGroup1.Network1.FBEstop2 Info Data/State
//     PlcTask Inputs/.STK_P2_050_SP01.PDOS.HwToPLC.EStop2State <-> Function Block Info Data/TwinSafeGroup1.Network1.FBEstop1 Info Data/State
//     PlcTask Outputs/.STK_P2_050_SP01.PDOS.PlcToHw.ErrorAcknowledgement <-> StandardOutputs/Standard In Var 1
//     PlcTask Outputs/.STK_P2_050_SP01.PDOS.PlcToHw.Run <-> StandardOutputs/Standard In Var 2
//     PlcTask Outputs/.STK_P2_050_SP01.PDOS.PlcToHw.safetyReset <-> StandardOutputs/Standard In Var 6
//   Plc_Program/Plc_Program Instance <-> NC-Task 1 SAF/Axes/Scorer1_Axis
//     PlcTask Inputs/.SLT1_P1_200_UG1.NcToPlc <-> Outputs/ToPlc
//     PlcTask Outputs/.SLT1_P1_200_UG1.PlcToNc <-> Inputs/FromPlc
//   Plc_Program/Plc_Program Instance <-> NC-Task 1 SAF/Axes/Scorer2_Axis
//     PlcTask Inputs/.SLT1_P1_200_UG2.NcToPlc <-> Outputs/ToPlc
//     PlcTask Outputs/.SLT1_P1_200_UG2.PlcToNc <-> Inputs/FromPlc
//   Plc_Program/Plc_Program Instance <-> NC-Task 1 SAF/Axes/Scorer3_Axis
//     PlcTask Inputs/.SLT1_P1_200_UG3.NcToPlc <-> Outputs/ToPlc
//     PlcTask Outputs/.SLT1_P1_200_UG3.PlcToNc <-> Inputs/FromPlc
//   Plc_Program/Plc_Program Instance <-> NC-Task 1 SAF/Axes/Scorer4_Axis
//     PlcTask Inputs/.SLT1_P1_200_UG4.NcToPlc <-> Outputs/ToPlc
//     PlcTask Outputs/.SLT1_P1_200_UG4.PlcToNc <-> Inputs/FromPlc
//   Plc_Program/Plc_Program Instance <-> NC-Task 1 SAF/Axes/Scorer5_Axis
//     PlcTask Inputs/.SLT1_P1_200_UG5.NcToPlc <-> Outputs/ToPlc
//     PlcTask Outputs/.SLT1_P1_200_UG5.PlcToNc <-> Inputs/FromPlc
//   Plc_Program/Plc_Program Instance <-> NC-Task 1 SAF/Axes/Scorer6_Axis
//     PlcTask Inputs/.SLT1_P1_200_UG6.NcToPlc <-> Outputs/ToPlc
//     PlcTask Outputs/.SLT1_P1_200_UG6.PlcToNc <-> Inputs/FromPlc
//   Plc_Program/Plc_Program Instance <-> NC-Task 1 SAF/Axes/Scorer7_Axis
//     PlcTask Inputs/.SLT1_P1_200_UG7.NcToPlc <-> Outputs/ToPlc
//     PlcTask Outputs/.SLT1_P1_200_UG7.PlcToNc <-> Inputs/FromPlc
//   Plc_Program/Plc_Program Instance <-> NC-Task 1 SAF/Axes/Scorer8_Axis
//     PlcTask Inputs/.SLT1_P1_200_UG8.NcToPlc <-> Outputs/ToPlc
//     PlcTask Outputs/.SLT1_P1_200_UG8.PlcToNc <-> Inputs/FromPlc
//   Plc_Program/Plc_Program Instance <-> NC-Task 1 SAF/Axes/knife1_Axis
//     PlcTask Inputs/.SLT1_P1_100_UG1.NcToPlc <-> Outputs/ToPlc
//     PlcTask Outputs/.SLT1_P1_100_UG1.PlcToNc <-> Inputs/FromPlc
//   Plc_Program/Plc_Program Instance <-> NC-Task 1 SAF/Axes/knife2_Axis
//     PlcTask Inputs/.SLT1_P1_100_UG2.NcToPlc <-> Outputs/ToPlc
//     PlcTask Outputs/.SLT1_P1_100_UG2.PlcToNc <-> Inputs/FromPlc
//   Plc_Program/Plc_Program Instance <-> NC-Task 1 SAF/Axes/knife3_Axis
//     PlcTask Inputs/.SLT1_P1_100_UG3.NcToPlc <-> Outputs/ToPlc
//     PlcTask Outputs/.SLT1_P1_100_UG3.PlcToNc <-> Inputs/FromPlc
//   Plc_Program/Plc_Program Instance <-> NC-Task 1 SAF/Axes/knife4_Axis
//     PlcTask Inputs/.SLT1_P1_100_UG4.NcToPlc <-> Outputs/ToPlc
//     PlcTask Outputs/.SLT1_P1_100_UG4.PlcToNc <-> Inputs/FromPlc
//   Plc_Program/Plc_Program Instance <-> NC-Task 1 SAF/Axes/knife5_Axis
//     PlcTask Inputs/.SLT1_P1_100_UG5.NcToPlc <-> Outputs/ToPlc
//     PlcTask Outputs/.SLT1_P1_100_UG5.PlcToNc <-> Inputs/FromPlc

CONFIGURATION Plc_Program
    RESOURCE PLC ON TwinCAT3
        TASK PlcFastTask(INTERVAL := T#5ms, PRIORITY := 1);
        TASK PlcTask(INTERVAL := T#20ms, PRIORITY := 20);
        PROGRAM FAST WITH PlcFastTask : FAST;
        PROGRAM MAIN WITH PlcTask : MAIN;
    END_RESOURCE
END_CONFIGURATION

// ---- Library/AxisControl/DataTypes/LAxisCtrl_typeAxisConfig.TcDUT
TYPE LAxisCtrl_typeAxisConfig :
STRUCT

  generalSettings 		: LAxisCtrl_typeGeneralSettings; 		(*Configuration of general settings*)
    power           			: LAxisCtrl_typePower;           			(*Configuration of MC_POWER function*)
    jog             			: LAxisCtrl_typeJog;             			(*Configuration of JOG function*)
    moveVelocity   	 	: LAxisCtrl_typeMoveVelocity;    		(*Configuration of MC_MOVEVELOCITY function*)
    stop            			: LAxisCtrl_typeStop;            			(*Configuration of MC_HALT function*)
    fastStop        			: LAxisCtrl_typeFastStop;        		(*Configuration of MC_HALT function (alternative dynamics)*)
    torqueLimiting  		: LAxisCtrl_typeTorqueLimiting; 		(*Configuration of MC_TORQUELIMITING function*)
    homing          			: LAxisCtrl_typeHoming;          		(*Configuration of HOMING function*)
    posRelative     		: LAxisCtrl_typePosRelative;     		(*Configuration of MC_MOVERELATIVE function*)
    posAbsolute     		: LAxisCtrl_typePosAbsolute;     		(*Configuration of MC_MOVEABSOLUTE function*)
    posSuperimposed		: LAxisCtrl_typePosSuperimposed; 	(*Configuration of MC_MOVESUPERIMPOSED function*)
    gearInRelative 	 	: LAxisCtrl_typeGearInRelative;  		(*Configuration of MC_GEARIN function*)
    gearInAbsolute 	 	: LAxisCtrl_typeGearInAbsolute;  		(*Configuration of MC_GEARIN_POS function*)
    camIn           			: LAxisCtrl_typeCamIn;           			(*Configuration of MC_CAMIN function*)
    phasing         			: LAxisCtrl_typePhasing;         		(*Configuration of MC_PHASING function*)

END_STRUCT
END_TYPE

// ---- Library/AxisControl/DataTypes/LAxisCtrl_typeCamIn.TcDUT
TYPE LAxisCtrl_typeCamIn :
STRUCT

	tableID				: INT := 1;
	masterOffset	    		: LREAL;		(*	Offset of leading values of cam	*)
	slaveOffset	            		: LREAL;		(*	Offset of following values of cam	*)
	masterScaling	        		: LREAL	:= 1;	(*	Scaling the leading values of the cam	*)
	slaveScaling	        		: LREAL	:= 1;	(*	Scaling the following values of the cam	*)
	masterStartPosition		: LREAL;		(*	Starting point in the cam/distance from the cam start with reference to the scaled cam	*)
	syncProfileReference		: DINT;		(*	Synchronization profile (0: Synchronization using dynamic parameters; 1: Synchronization using leading value distance; 2: Direct synchronous setting)	*)
	masterStartDistance		: LREAL;		(*	Leading value distance (when "SyncProfileReference" = 1)	*)
	velocity	            		: LREAL;		(*	Velocity for synchronization (when "SyncProfileReference" = 0; Value > 0.0: The specified value is used; Value = 0.0: Not permitted; Value < 0.0: Use of the default value configured in the technology object)	*)
	acceleration	        		: LREAL;		(*	Acceleration for synchronization (when "SyncProfileReference" = 0; Value > 0.0: The specified value is used; Value = 0.0: Not permitted; Value < 0.0: Use of the default value configured in the technology object)	*)
	deceleration	        		: LREAL;		(*	Deceleration for synchronization (when "SyncProfileReference" = 0; Value > 0.0: The specified value is used; Value = 0.0: Not permitted; Value < 0.0: Use of the default value configured in the technology object)	*)
	jerk	                			: LREAL;		(*	Jerk for synchronization (when "SyncProfileReference" = 0; Value > 0.0: Smooth velocity profile, the specified value is used; Value = 0.0: Trapezoid velocity profile; Value < 0.0: Use of the default value configured in the technology object)	*)
	applicationMode	        		:  DINT;		(*	Application of the cam (0: Once/not cyclic; 1: Cyclic ; 2: Cyclic appending)	*)
	syncDirection	        		: DINT;		(*	Direction for synchronization only in effect for axes with activated modulo setting (1: Forward direction; 2: Backward direction; 3: Shortest way)	*)
	ActivationPosition		: LREAL;
//	startMode				: MC_StartMode  := MC_STARTMODE_ABSOLUTE;
//	ActivationMode			: MC_CamActivationMode;

END_STRUCT
END_TYPE

// ---- Library/AxisControl/DataTypes/LAxisCtrl_typeDiagnostics.TcDUT
TYPE LAxisCtrl_typeDiagnostics :
STRUCT

	status						:WORD;	(*Status OF FB when error occurred*)
	subfunctionStatus			:UDINT;	(*ErrorID OF called subfunction*)
	basicMotionState			:DINT;	(*Current basic motion state when error occurred*)
	superimposedMotionState		:DINT;	(*Current superimposed motion state when error occurred*)

END_STRUCT
END_TYPE

// ---- Library/AxisControl/DataTypes/LAxisCtrl_typeFastStop.TcDUT
TYPE LAxisCtrl_typeFastStop :
STRUCT

	deceleration			: LREAL;	(*Deceleration FOR fast stop (Value > 0.0: The specified value is used; Value <= 0.0: emergency deceleration OF  the technology object is used)*)
	jerk					: LREAL;	(*Jerk FOR fast stop (Value > 0.0: Smooth velocity profile, the specified value is used; Value = 0.0: Trapezoid velocity profile; Value < 0.0: Use OF the default value configured in the technology object)*)
	abortAcceleration		: BOOL;	(*The acceleration is set TO 0.0 AT the start OF the job, AND the deceleration immediately builds up; FALSE: The current acceleration AT the start OF the job is reduced using the configured jerk. Afterwards, the deceleration builds up*)
	replaceStopPossible		: BOOL;	(*Fast stop command can be replaced BY another command*)

END_STRUCT
END_TYPE

// ---- Library/AxisControl/DataTypes/LAxisCtrl_typeGearInAbsolute.TcDUT
TYPE LAxisCtrl_typeGearInAbsolute :
STRUCT

	ratioNumerator			       	:DINT;	(*Gear ratio numerator*)
	ratioDenominator			   	:DINT;	(*Gear ratio denominator*)
	masterSyncPosition		        	:LREAL;	(*Synchronous position of leading axis*)
	slaveSyncPosition		        	:LREAL;	(*Synchronous position of following axis*)
	syncProfileReference	        		:DINT;	(*Type of synchronization (0: Synchronization using dynamic parameters; 1: Synchronization using leading value distance)*)
	masterStartDistance	            	:LREAL;	(*Leading value distance (when "SyncProfileReference" = 1)*)
	velocity					:LREAL;	(*Velocity for synchronization (when "SyncProfileReference" = 0; Value > 0.0: The specified value is used; Value = 0.0: Not permitted; Value < 0.0: Use of the default value configured in the technology object)*)
	acceleration			  	:LREAL;	(*Acceleration for synchronization (when "SyncProfileReference" = 0; Value > 0.0: The specified value is used; Value = 0.0: Not permitted; Value < 0.0: Use of the default value configured in the technology object)*)
	deceleration			    	:LREAL;	(*Deceleration for synchronization (when "SyncProfileReference" = 0; Value > 0.0: The specified value is used; Value = 0.0: Not permitted; Value < 0.0: Use of the default value configured in the technology object)*)
	jerk						:LREAL;	(*Jerk for synchronization (when "SyncProfileReference" = 0; Value > 0.0: Smooth velocity profile, the specified value is used; Value = 0.0: Trapezoid velocity profile; Value < 0.0: Use of the default value configured in the technology object)*)
	syncDirection			    	:DINT;	(*Direction for synchronization only in effect for axes with activated modulo setting (1: Forward direction; 2: Backward direction; 3: Shortest way)*)
	ratioChangeOnTheFly	            	:BOOL;	(*TRUE: Changing gear ratio on-the-fly; FALSE: Ratio change requires a new rising edge at gearInAbsolute input*)

END_STRUCT
END_TYPE

// ---- Library/AxisControl/DataTypes/LAxisCtrl_typeGearInRelative.TcDUT
TYPE LAxisCtrl_typeGearInRelative :
STRUCT

	ratioNumerator       		: DINT  	:= 1;      	 (* Gear ratio numerator*)
      	ratioDenominator    		: DINT  	:= 1;      	 (* Gear ratio denominator*)
      	acceleration        			: LREAL 	:= -1.0;	 (*Acceleration for synchronization (when "SyncProfileReference"  = 0; Value > 0.0: The specified value is used; Value = 0.0: Not permitted; Value < 0.0: Use of the default value configured in the technology object)*)
      	deceleration        			: LREAL 	:= -1.0; 	 (* Deceleration for synchronization (when "SyncProfileReference" = 0; Value > 0.0: The specified value is used; Value = 0.0: Not permitted; Value < 0.0: Use of the default value configured in the technology object)*)
      	jerk                			: LREAL 	:= -1.0;   	 (*Jerk for synchronization (when "SyncProfileReference"          = 0; Value > 0.0: Smooth velocity profile, the specified value is used; Value = 0.0: Trapezoid velocity profile; Value < 0.0: Use of the default value configured in the technology object)*)
      	ratioChangeOnTheFly 		: BOOL 	:= FALSE;   (* TRUE: Changing gear ratio on-the-fly; FALSE: Ratio change requires a NE*)

END_STRUCT
END_TYPE

// ---- Library/AxisControl/DataTypes/LAxisCtrl_typeGeneralSettings.TcDUT
TYPE LAxisCtrl_typeGeneralSettings :
STRUCT

	stopOnError			:BOOL;
	resetWithRestart			:BOOL;
	abortWaitingSyncCmd		:BOOL;

END_STRUCT
END_TYPE

// ---- Library/AxisControl/DataTypes/LAxisCtrl_typeHoming.TcDUT
TYPE LAxisCtrl_typeHoming :
STRUCT

	position					: LREAL	:= 00.0;	(*The specified value is used according to the selected "Mode"*)
	offsetPosition				: LREAL	:= 200;	(*Homing offset postion*)
	offsetPositionVelocity			: LREAL	:= 100.0;	(*Homing offset execution velocicy*)
	offsetPositionAcceleration		: LREAL	:= 100.0;	(*Homing offset execution acceleration*)
	offsetPositonDeceleration		: LREAL	:= 100.0;	(*Homing offset execution deceleration*)
	offsetPositionJerk			: LREAL	:= 100.0;	(*Homing offset execution Jerk*)
	mode						: INT		:= 0;		(*-1: Standard homming using MC_HOME; Operation mode; 0: Direct homing (absolute); 1:Direct homing (relative); 2:Passive homing (without reset); 3:Active homing; 5:Active homing (Position parameter has no effect); 6:Absolute encoder adjustment (relative); 7:Absolute encoder adjustment (absolute); 8:Passive homing ; 9:Abort passive homing; 10: Passive homing (Position parameter has no effect)*)
	extendedMode				: DINT	:= 0;		(*-1: No extended homing mode (parameter "mode" is effective); 0: Homing on fixed stop;*)
	extendedModeTorqueLimit		: LREAL	:= 100.0;	(* Value of the torque/force for extended homing mode*)
	homeExecutionTimeLimit		: TIME	:= T#2M;	(*Home execution maximum time*)

END_STRUCT
END_TYPE

// ---- Library/AxisControl/DataTypes/LAxisCtrl_typeJog.TcDUT
TYPE LAxisCtrl_typeJog :
STRUCT
	velocity			:LREAL;
	acceleration		:LREAL;
	deceleration		:LREAL;
	jerk				:LREAL;
	positionControlled	:BOOL;
	increment			:LREAL;
	mode				:DINT;

END_STRUCT
END_TYPE

// ---- Library/AxisControl/DataTypes/LAxisCtrl_typeMoveVelocity.TcDUT
TYPE LAxisCtrl_typeMoveVelocity :
STRUCT

	 velocity               			: LREAL := 100;     			(* Velocity/Speed FOR motion process (Value = 0.0: Permitted)*)
      	acceleration           		: LREAL := 100;    				(* Acceleration setpoint for motion process (Value > 0.0: The specified value is used; Value = 0.0: Not permitted; Value < 0.0: Use of the default value configured in the technology object)*)
      	deceleration           		: LREAL := 100;    				(* Deceleration setpoint for motion process (Value > 0.0: The specified value is used; Value = 0.0: Not permitted; Value < 0.0: Use of the default value configured in the technology object)*)
      	jerk                  			: LREAL := 100;   	 			(* Jerk for velocity specification (Value > 0.0: Smooth velocity profile, the specified value is used; (Value = 0.0: Trapezoid velocity profile; (Value < 0.0: Use of the default value configured in the technology object)*)
      	direction            			: INT   := MC_Positive_Direction ;	(* Motion direction of the axis (0: Not Used (Error); 1: Positive direction; 3: Negative direction)*)
      	positionControlled     		: BOOL  := FALSE;   			(* TRUE: Position-controlled operation; FALSE: Non position-controlled operation*)
      	velocityChangeOnTheFly 	: BOOL  := TRUE;  			(* TRUE: Changing velocity on-the-fly; FALSE: Velocity change requires a new rising edge on moveVelocity input*)

END_STRUCT
END_TYPE

// ---- Library/AxisControl/DataTypes/LAxisCtrl_typePhasing.TcDUT
TYPE LAxisCtrl_typePhasing :
STRUCT

	phaseShift               		: LREAL;
	velocity                 		: LREAL;
 	acceleration			: LREAL;
	deceleration			: LREAL;
	jerk                     			: LREAL;
	phaseAbsolute            		: BOOL;
	phaseShiftChangeOnTheFly 	: BOOL;

END_STRUCT
END_TYPE

// ---- Library/AxisControl/DataTypes/LAxisCtrl_typePosAbsolute.TcDUT
TYPE LAxisCtrl_typePosAbsolute :
STRUCT

 	position				: LREAL := 0.0;    (* Absolute target position*)
      	velocity				: LREAL := 100;    (*Velocity setpoint for absolute positioning (Value > 0.0: The specified value is used; Value = 0.0: Not permitted; Value < 0.0: Use of the default value configured in the technology object)*)
      	acceleration			: LREAL := 100;   (* Acceleration setpoint for absolute positioning (Value > 0.0: The specified value is used; Value = 0.0: Not permitted; Value < 0.0: Use of the default value configured in the technology object)*)
      	deceleration			: LREAL := 100;    (* Deceleration setpoint for absolute positioning (Value > 0.0: The specified value is used; Value = 0.0: Not permitted; Value < 0.0: Use of the default value configured in the technology object)*)
      	jerk					: LREAL := 100;    (* Jerk for absolute positioning (Value > 0.0: Smooth velocity profile, the specified value is used; (Value = 0.0: Trapezoid velocity profile; (Value < 0.0: Use of the default value configured in the technology object)*)
      	direction				: INT   := 1;      (* Motion direction of the axis (1: Positive direction; 2: Negative direction; 3: Shortest way)*)
      	positionChangeOnTheFly	: BOOL  := TRUE;   (* TRUE: Changing position on-the-fly; FALSE: Position change requires a new rising edge at posAbsolute input*)
      	velocityChangeOnTheFly	: BOOL  := TRUE;   (* TRUE: Changing velocity on-the-fly; FALSE: Velocity change requires a new rising edge at posAbsolute input*)


END_STRUCT
END_TYPE

// ---- Library/AxisControl/DataTypes/LAxisCtrl_typePosRelative.TcDUT
TYPE LAxisCtrl_typePosRelative :
STRUCT

 	distance    		: LREAL := 200.0;    	(* Distance FOR positioning process*)
	velocity     		: LREAL := 100;      	(* Velocity setpoint for relative positioning (Value > 0.0: The specified value is used; Value = 0.0: Not permitted; Value < 0.0: Use of the default value configured in the technology object)*)
      	acceleration 	: LREAL := 100;     	(* Acceleration setpoint for relative positioning (Value > 0.0: The specified value is used; Value = 0.0: Not permitted; Value < 0.0: Use of the default value configured in the technology object)*)
      	deceleration 	: LREAL := 100;      	(* Deceleration setpoint for relative positioning (Value > 0.0: The specified value is used; Value = 0.0: Not permitted; Value < 0.0: Use of the default value configured in the technology object)*)
      	jerk         		: LREAL := 100;      	(* Jerk for relative positioning (Value > 0.0: Smooth velocity profile, the specified value is used; Value = 0.0: Trapezoid velocity profile; Value < 0.0: Use of the default value configured in the technology object)*)
      	direction    		: DINT  := 1;        		(* Motion direction of the axis (0: The sign of the distance parameter defines the direction; 1: Positive direction; 2: Negative direction)*)



END_STRUCT
END_TYPE

// ---- Library/AxisControl/DataTypes/LAxisCtrl_typePosSuperimposed.TcDUT
TYPE LAxisCtrl_typePosSuperimposed :
STRUCT

	distance		: LREAL;
	velocityDiff		: LREAL;
	acceleration	: LREAL;
	deceleration	: LREAL;
	jerk			: LREAL;
	direction		: DINT;

END_STRUCT
END_TYPE

// ---- Library/AxisControl/DataTypes/LAxisCtrl_typePower.TcDUT
TYPE LAxisCtrl_typePower :
STRUCT

	startMode			: DINT;
	stopMode			: INT;
	syncMotionSimulation	: BOOL;

END_STRUCT
END_TYPE

// ---- Library/AxisControl/DataTypes/LAxisCtrl_typeStop.TcDUT
TYPE LAxisCtrl_typeStop :
STRUCT

	deceleration		: LREAL;
	jerk				: REAL;
	abortAcceleration	: BOOL;

END_STRUCT
END_TYPE

// ---- Library/AxisControl/DataTypes/LAxisCtrl_typeTorqueLimiting.TcDUT
TYPE LAxisCtrl_typeTorqueLimiting :
STRUCT

	TorqueLimit	: LREAL;
	mode			: DINT;

END_STRUCT
END_TYPE

// ---- Library/AxisControl/DataTypes/LRK_typeCamCommand.TcDUT
TYPE LRK_typeCamCommand :
STRUCT
	
	resetExecute:BOOL;
	resetRestart:BOOL;
	interpolateCamExecute:BOOL;

END_STRUCT
END_TYPE

// ---- Library/AxisControl/DataTypes/LRK_typeCamStatus.TcDUT
TYPE
LRK_typeCamStatus :
STRUCT
    cam                      : INT;
    control                  : BOOL;
    error                    : BOOL;
    restartActive            : BOOL;
    onlineStartValuesChanged : BOOL;
    camDataChanged           : BOOL;
    interpolated             : BOOL;
    inInterpolation          : BOOL;
    restartDone              : BOOL;
    restartBusy              : BOOL;
    restartCommandAborted    : BOOL;
    restartError             : BOOL;
    restartErrorId           : WORD;
    interpolateCamDone       : BOOL;
    interpolateCamBusy       : BOOL;
    interpolateCamError      : BOOL;
    interpolateCamErrorId    : WORD;
    startLeadingValue        : LREAL;
    endLeadingValue          : LREAL;
END_STRUCT
END_TYPE

// ---- Library/AxisControl/DataTypes/LRK_typeRotaryKnifeAxisCommand.TcDUT
TYPE LRK_typeRotaryKnifeAxisCommand :
STRUCT

	enable 			: BOOL;
      	resetAxis 			: BOOL;
  	enableAxis 		: BOOL;
	jogForward 		: BOOL;
      	jogBackward 		: BOOL;
      	moveVelocity 		: BOOL;
      	posAbsolute 		: BOOL;
      	posRelative 		: BOOL;
      	posSuperimposed 	: BOOL;
      	homing 			: BOOL;
      	stop 				: BOOL;
      	fastStop 			: BOOL;
      	torqueLimiting 		: BOOL;
      	gearInRelative 		: BOOL;
      	gearInAbsolute 		: BOOL;
      	camIn 			: BOOL;
      	phasing 			: BOOL;

END_STRUCT
END_TYPE

// ---- Library/AxisControl/DataTypes/LRK_typeUsersInterface.TcDUT
TYPE LRK_typeUsersInterface:
STRUCT

